LIN {X 0,Y 319.575,Z 275.493,A -85,B 0,C 180,E1 -15365.301,E2 -15365.301} C_VEL
LIN {X 0,Y 319.566,Z 275.493,A -85,B 0,C 180,E1 -15368.045,E2 -15368.045} C_VEL
LIN {X 0,Y 319.59,Z 275.527,A -85,B 0,C 180,E1 -15370.003,E2 -15370.003} C_VEL
LIN {X 0,Y 319.829,Z 276.598,A -85,B 0,C 180,E1 -15370.301,E2 -15370.301} C_VEL
LIN {X 0,Y 325.235,Z 292.198,A -85,B 0,C 180,E1 -15371.007,E2 -15371.007} C_VEL
LIN {X 0,Y 326.367,Z 298.329,A -85,B 0,C 180,E1 -15371.217,E2 -15371.217} C_VEL
LIN {X 0,Y 325.364,Z 352.937,A -85,B 0,C 180,E1 -15372.438,E2 -15372.438} C_VEL
LIN {X 0,Y 325.113,Z 362.734,A -85,B 0,C 180,E1 -15372.829,E2 -15372.829} C_VEL
LIN {X 0,Y 324.671,Z 373.811,A -85,B 0,C 180,E1 -15373.494,E2 -15373.494} C_VEL
LIN {X 0,Y 323.823,Z 384.617,A -85,B 0,C 180,E1 -15374.42,E2 -15374.42} C_VEL
LIN {X 0,Y 323.214,Z 391.764,A -85,B 0,C 180,E1 -15375.197,E2 -15375.197} C_VEL
LIN {X 0,Y 322.423,Z 399.87,A -85,B 0,C 180,E1 -15376.287,E2 -15376.287} C_VEL
LIN {X 0,Y 321.691,Z 406.556,A -85,B 0,C 180,E1 -15377.38,E2 -15377.38} C_VEL
LIN {X 0,Y 320.885,Z 412.887,A -85,B 0,C 180,E1 -15378.631,E2 -15378.631} C_VEL
LIN {X 0,Y 320.082,Z 419.308,A -85,B 0,C 180,E1 -15380.202,E2 -15380.202} C_VEL
LIN {X 0,Y 319.481,Z 424.66,A -85,B 0,C 180,E1 -15381.858,E2 -15381.858} C_VEL
LIN {X 0,Y 318.896,Z 429.161,A -85,B 0,C 180,E1 -15383.673,E2 -15383.673} C_VEL
LIN {X 0,Y 318.57,Z 431.47,A -85,B 0,C 180,E1 -15384.937,E2 -15384.937} C_VEL
LIN {X 0,Y 318.385,Z 433.223,A -85,B 0,C 180,E1 -15386.202,E2 -15386.202} C_VEL
LIN {X 0,Y 318.229,Z 434.488,A -85,B 0,C 180,E1 -15387.468,E2 -15387.468} C_VEL
LIN {X 0,Y 318.122,Z 435.287,A -85,B 0,C 180,E1 -15388.733,E2 -15388.733} C_VEL
LIN {X 0,Y 318.09,Z 435.591,A -85,B 0,C 180,E1 -15389.999,E2 -15389.999} C_VEL
LIN {X 0,Y 318.121,Z 435.315,A -85,B 0,C 180,E1 -15391.265,E2 -15391.265} C_VEL
LIN {X 0,Y 318.212,Z 434.573,A -85,B 0,C 180,E1 -15392.531,E2 -15392.531} C_VEL
LIN {X 0,Y 318.378,Z 433.365,A -85,B 0,C 180,E1 -15393.796,E2 -15393.796} C_VEL
LIN {X 0,Y 318.699,Z 430.531,A -85,B 0,C 180,E1 -15395.694,E2 -15395.694} C_VEL
LIN {X 0,Y 319.1,Z 427.945,A -85,B 0,C 180,E1 -15396.957,E2 -15396.957} C_VEL
LIN {X 0,Y 319.589,Z 424,A -85,B 0,C 180,E1 -15398.472,E2 -15398.472} C_VEL
LIN {X 0,Y 320.185,Z 418.558,A -85,B 0,C 180,E1 -15400.113,E2 -15400.113} C_VEL
LIN {X 0,Y 320.841,Z 413.383,A -85,B 0,C 180,E1 -15401.369,E2 -15401.369} C_VEL
LIN {X 0,Y 321.669,Z 407.142,A -85,B 0,C 180,E1 -15402.619,E2 -15402.619} C_VEL
LIN {X 0,Y 322.491,Z 399.559,A -85,B 0,C 180,E1 -15403.869,E2 -15403.869} C_VEL
LIN {X 0,Y 323.354,Z 390.109,A -85,B 0,C 180,E1 -15405.118,E2 -15405.118} C_VEL
LIN {X 0,Y 324.216,Z 380.839,A -85,B 0,C 180,E1 -15406.044,E2 -15406.044} C_VEL
LIN {X 0,Y 324.812,Z 371.887,A -85,B 0,C 180,E1 -15406.74,E2 -15406.74} C_VEL
LIN {X 0,Y 325.173,Z 362.547,A -85,B 0,C 180,E1 -15407.288,E2 -15407.288} C_VEL
LIN {X 0,Y 325.397,Z 353.548,A -85,B 0,C 180,E1 -15407.652,E2 -15407.652} C_VEL
LIN {X 0,Y 326.401,Z 302.241,A -85,B 0,C 180,E1 -15408.803,E2 -15408.803} C_VEL
LIN {X 0,Y 326.205,Z 297.195,A -85,B 0,C 180,E1 -15408.93,E2 -15408.93} C_VEL
LIN {X 0,Y 324.486,Z 289.724,A -85,B 0,C 180,E1 -15409.208,E2 -15409.208} C_VEL
LIN {X 0,Y 319.743,Z 276.336,A -85,B 0,C 180,E1 -15409.844,E2 -15409.844} C_VEL
LIN {X 0,Y 319.588,Z 275.493,A -85,B 0,C 180,E1 -15410.18,E2 -15410.18} C_VEL
LIN {X 0,Y 319.541,Z 275.494,A -85,B 0,C 180,E1 -15413.321,E2 -15413.321} C_VEL
LIN {X 0,Y 319.548,Z 275.494,A -85,B 0,C 180,E1 -15416.095,E2 -15416.095} C_VEL
LIN {X 0,Y 319.522,Z 275.496,A -85,B 0,C 180,E1 -15418.939,E2 -15418.939} C_VEL
LIN {X 0,Y 319.517,Z 275.496,A -85,B 0,C 180,E1 -15421.862,E2 -15421.862} C_VEL
LIN {X 0,Y 319.576,Z 275.487,A -85,B 0,C 180,E1 -15425.542,E2 -15425.542} C_VEL
LIN {X 0,Y 319.525,Z 275.495,A -85,B 0,C 180,E1 -15429.661,E2 -15429.661} C_VEL
LIN {X 0,Y 319.515,Z 275.495,A -85,B 0,C 180,E1 -15433.459,E2 -15433.459} C_VEL
LIN {X 0,Y 319.475,Z 275.497,A -85,B 0,C 180,E1 -15434.327,E2 -15434.327} C_VEL
LIN {X 0,Y 318.821,Z 275.583,A -85,B 0,C 180,E1 -15435.38,E2 -15435.38} C_VEL
LIN {X 0,Y 316.003,Z 275.942,A -85,B 0,C 180,E1 -15437.095,E2 -15437.095} C_VEL
LIN {X 0,Y 313.597,Z 276.243,A -85,B 0,C 180,E1 -15438.484,E2 -15438.484} C_VEL
LIN {X 0,Y 312.545,Z 276.369,A -85,B 0,C 180,E1 -15439.559,E2 -15439.559} C_VEL
LIN {X 0,Y 312.449,Z 276.378,A -85,B 0,C 180,E1 -15439.923,E2 -15439.923} C_VEL
LIN {X 0,Y 312.529,Z 276.366,A -85,B 0,C 180,E1 -15444.05,E2 -15444.05} C_VEL
LIN {X 0,Y 312.497,Z 276.371,A -85,B 0,C 180,E1 -15447.333,E2 -15447.333} C_VEL
LIN {X 0,Y 312.493,Z 276.373,A -85,B 0,C 180,E1 -15451.294,E2 -15451.294} C_VEL
LIN {X 0,Y 312.542,Z 276.364,A -85,B 0,C 180,E1 -15454.707,E2 -15454.707} C_VEL
LIN {X 0,Y 312.536,Z 276.367,A -85,B 0,C 180,E1 -15457.525,E2 -15457.525} C_VEL
LIN {X 0,Y 312.546,Z 276.363,A -85,B 0,C 180,E1 -15461.651,E2 -15461.651} C_VEL
LIN {X 0,Y 312.646,Z 276.346,A -85,B 0,C 180,E1 -15465.684,E2 -15465.684} C_VEL
LIN {X 0,Y 312.679,Z 276.346,A -85,B 0,C 180,E1 -15469.641,E2 -15469.641} C_VEL
LIN {X 0,Y 312.79,Z 276.333,A -85,B 0,C 180,E1 -15472.252,E2 -15472.252} C_VEL
LIN {X 0,Y 312.68,Z 276.345,A -85,B 0,C 180,E1 -15474.842,E2 -15474.842} C_VEL
LIN {X 0,Y 312.961,Z 276.313,A -85,B 0,C 180,E1 -15478.713,E2 -15478.713} C_VEL
LIN {X 0,Y 312.961,Z 276.311,A -85,B 0,C 180,E1 -15481.287,E2 -15481.287} C_VEL
LIN {X 0,Y 312.68,Z 276.345,A -85,B 0,C 180,E1 -15485.158,E2 -15485.158} C_VEL
LIN {X 0,Y 312.79,Z 276.333,A -85,B 0,C 180,E1 -15487.748,E2 -15487.748} C_VEL
LIN {X 0,Y 312.654,Z 276.349,A -85,B 0,C 180,E1 -15491.672,E2 -15491.672} C_VEL
LIN {X 0,Y 312.609,Z 276.355,A -85,B 0,C 180,E1 -15494.828,E2 -15494.828} C_VEL
LIN {X 0,Y 312.529,Z 276.365,A -85,B 0,C 180,E1 -15499.186,E2 -15499.186} C_VEL
LIN {X 0,Y 312.508,Z 276.368,A -85,B 0,C 180,E1 -15502.775,E2 -15502.775} C_VEL
LIN {X 0,Y 312.476,Z 276.372,A -85,B 0,C 180,E1 -15506.732,E2 -15506.732} C_VEL
LIN {X 0,Y 312.463,Z 276.379,A -85,B 0,C 180,E1 -15509.658,E2 -15509.658} C_VEL
LIN {X 0,Y 312.515,Z 276.372,A -85,B 0,C 180,E1 -15513.689,E2 -15513.689} C_VEL
LIN {X 0,Y 312.505,Z 276.374,A -85,B 0,C 180,E1 -15517.388,E2 -15517.388} C_VEL
LIN {X 0,Y 312.436,Z 276.378,A -85,B 0,C 180,E1 -15520.718,E2 -15520.718} C_VEL
LIN {X 0,Y 312.445,Z 276.376,A -85,B 0,C 180,E1 -15524.211,E2 -15524.211} C_VEL
LIN {X 0,Y 312.449,Z 276.376,A -85,B 0,C 180,E1 -15527.926,E2 -15527.926} C_VEL
LIN {X 0,Y 312.479,Z 276.372,A -85,B 0,C 180,E1 -15531.923,E2 -15531.923} C_VEL
LIN {X 0,Y 312.526,Z 276.366,A -85,B 0,C 180,E1 -15534.221,E2 -15534.221} C_VEL
LIN {X 0,Y 312.496,Z 276.371,A -85,B 0,C 180,E1 -15537.334,E2 -15537.334} C_VEL
LIN {X 0,Y 312.553,Z 276.446,A -85,B 0,C 180,E1 -15540.259,E2 -15540.259} C_VEL
LIN {X 0,Y 314.554,Z 286.634,A -85,B 0,C 180,E1 -15543.459,E2 -15543.459} C_VEL
LIN {X 0,Y 315.392,Z 291.548,A -85,B 0,C 180,E1 -15544.952,E2 -15544.952} C_VEL
LIN {X 0,Y 314.713,Z 298.783,A -85,B 0,C 180,E1 -15546.997,E2 -15546.997} C_VEL
LIN {X 0,Y 313.718,Z 308.843,A -85,B 0,C 180,E1 -15549.813,E2 -15549.813} C_VEL
LIN {X 0,Y 317.665,Z 337.125,A -85,B 0,C 180,E1 -15550.735,E2 -15550.735} C_VEL
LIN {X 0,Y 318.865,Z 349.16,A -85,B 0,C 180,E1 -15551.089,E2 -15551.089} C_VEL
LIN {X 0,Y 318.114,Z 387.635,A -85,B 0,C 180,E1 -15551.984,E2 -15551.984} C_VEL
LIN {X 0,Y 317.516,Z 398.812,A -85,B 0,C 180,E1 -15552.448,E2 -15552.448} C_VEL
LIN {X 0,Y 316.588,Z 410.517,A -85,B 0,C 180,E1 -15553.227,E2 -15553.227} C_VEL
LIN {X 0,Y 315.722,Z 419.221,A -85,B 0,C 180,E1 -15554.011,E2 -15554.011} C_VEL
LIN {X 0,Y 314.88,Z 427.545,A -85,B 0,C 180,E1 -15554.962,E2 -15554.962} C_VEL
LIN {X 0,Y 313.925,Z 435.427,A -85,B 0,C 180,E1 -15556.075,E2 -15556.075} C_VEL
LIN {X 0,Y 313.015,Z 442.804,A -85,B 0,C 180,E1 -15557.356,E2 -15557.356} C_VEL
LIN {X 0,Y 312.134,Z 450.298,A -85,B 0,C 180,E1 -15558.967,E2 -15558.967} C_VEL
LIN {X 0,Y 311.431,Z 457.151,A -85,B 0,C 180,E1 -15560.912,E2 -15560.912} C_VEL
LIN {X 0,Y 311.013,Z 462.366,A -85,B 0,C 180,E1 -15562.861,E2 -15562.861} C_VEL
LIN {X 0,Y 310.798,Z 466.2,A -85,B 0,C 180,E1 -15564.811,E2 -15564.811} C_VEL
LIN {X 0,Y 310.82,Z 467.97,A -85,B 0,C 180,E1 -15566.111,E2 -15566.111} C_VEL
LIN {X 0,Y 310.8,Z 469.234,A -85,B 0,C 180,E1 -15567.409,E2 -15567.409} C_VEL
LIN {X 0,Y 310.872,Z 470.023,A -85,B 0,C 180,E1 -15568.705,E2 -15568.705} C_VEL
LIN {X 0,Y 310.987,Z 470.326,A -85,B 0,C 180,E1 -15570.001,E2 -15570.001} C_VEL
LIN {X 0,Y 310.872,Z 470.018,A -85,B 0,C 180,E1 -15571.296,E2 -15571.296} C_VEL
LIN {X 0,Y 310.801,Z 469.217,A -85,B 0,C 180,E1 -15572.593,E2 -15572.593} C_VEL
LIN {X 0,Y 310.821,Z 467.941,A -85,B 0,C 180,E1 -15573.89,E2 -15573.89} C_VEL
LIN {X 0,Y 310.844,Z 464.997,A -85,B 0,C 180,E1 -15575.838,E2 -15575.838} C_VEL
LIN {X 0,Y 311.011,Z 462.314,A -85,B 0,C 180,E1 -15577.14,E2 -15577.14} C_VEL
LIN {X 0,Y 311.431,Z 457.083,A -85,B 0,C 180,E1 -15579.09,E2 -15579.09} C_VEL
LIN {X 0,Y 312.13,Z 450.197,A -85,B 0,C 180,E1 -15581.034,E2 -15581.034} C_VEL
LIN {X 0,Y 313.007,Z 442.688,A -85,B 0,C 180,E1 -15582.646,E2 -15582.646} C_VEL
LIN {X 0,Y 313.919,Z 435.29,A -85,B 0,C 180,E1 -15583.927,E2 -15583.927} C_VEL
LIN {X 0,Y 314.899,Z 427.377,A -85,B 0,C 180,E1 -15585.038,E2 -15585.038} C_VEL
LIN {X 0,Y 315.776,Z 419.013,A -85,B 0,C 180,E1 -15585.988,E2 -15585.988} C_VEL
LIN {X 0,Y 316.758,Z 408.327,A -85,B 0,C 180,E1 -15586.931,E2 -15586.931} C_VEL
LIN {X 0,Y 317.576,Z 396.677,A -85,B 0,C 180,E1 -15587.633,E2 -15587.633} C_VEL
LIN {X 0,Y 318.137,Z 386.897,A -85,B 0,C 180,E1 -15588.016,E2 -15588.016} C_VEL
LIN {X 0,Y 318.747,Z 347.007,A -85,B 0,C 180,E1 -15588.945,E2 -15588.945} C_VEL
LIN {X 0,Y 315.503,Z 321.052,A -85,B 0,C 180,E1 -15589.755,E2 -15589.755} C_VEL
LIN {X 0,Y 313.72,Z 308.721,A -85,B 0,C 180,E1 -15590.199,E2 -15590.199} C_VEL
LIN {X 0,Y 315.293,Z 293.881,A -85,B 0,C 180,E1 -15594.354,E2 -15594.354} C_VEL
LIN {X 0,Y 315.204,Z 290.232,A -85,B 0,C 180,E1 -15595.418,E2 -15595.418} C_VEL
LIN {X 0,Y 313.077,Z 279,A -85,B 0,C 180,E1 -15598.899,E2 -15598.899} C_VEL
LIN {X 0,Y 312.556,Z 276.361,A -85,B 0,C 180,E1 -15599.742,E2 -15599.742} C_VEL
LIN {X 0,Y 312.506,Z 276.367,A -85,B 0,C 180,E1 -15604.211,E2 -15604.211} C_VEL
LIN {X 0,Y 312.513,Z 276.37,A -85,B 0,C 180,E1 -15607.388,E2 -15607.388} C_VEL
LIN {X 0,Y 312.441,Z 276.38,A -85,B 0,C 180,E1 -15610.718,E2 -15610.718} C_VEL
LIN {X 0,Y 312.45,Z 276.376,A -85,B 0,C 180,E1 -15614.21,E2 -15614.21} C_VEL
LIN {X 0,Y 312.454,Z 276.375,A -85,B 0,C 180,E1 -15617.925,E2 -15617.925} C_VEL
LIN {X 0,Y 312.476,Z 276.373,A -85,B 0,C 180,E1 -15621.925,E2 -15621.925} C_VEL
LIN {X 0,Y 312.531,Z 276.368,A -85,B 0,C 180,E1 -15624.22,E2 -15624.22} C_VEL
LIN {X 0,Y 312.502,Z 276.368,A -85,B 0,C 180,E1 -15627.334,E2 -15627.334} C_VEL
LIN {X 0,Y 312.485,Z 276.37,A -85,B 0,C 180,E1 -15631.3,E2 -15631.3} C_VEL
LIN {X 0,Y 312.516,Z 276.368,A -85,B 0,C 180,E1 -15634.705,E2 -15634.705} C_VEL
LIN {X 0,Y 312.54,Z 276.364,A -85,B 0,C 180,E1 -15637.526,E2 -15637.526} C_VEL
LIN {X 0,Y 312.54,Z 276.366,A -85,B 0,C 180,E1 -15641.651,E2 -15641.651} C_VEL
LIN {X 0,Y 312.638,Z 276.354,A -85,B 0,C 180,E1 -15645.684,E2 -15645.684} C_VEL
LIN {X 0,Y 312.683,Z 276.348,A -85,B 0,C 180,E1 -15649.641,E2 -15649.641} C_VEL
LIN {X 0,Y 312.841,Z 276.324,A -85,B 0,C 180,E1 -15653.551,E2 -15653.551} C_VEL
LIN {X 0,Y 312.967,Z 276.31,A -85,B 0,C 180,E1 -15658.713,E2 -15658.713} C_VEL
LIN {X 0,Y 312.968,Z 276.313,A -85,B 0,C 180,E1 -15661.287,E2 -15661.287} C_VEL
LIN {X 0,Y 312.686,Z 276.343,A -85,B 0,C 180,E1 -15665.158,E2 -15665.158} C_VEL
LIN {X 0,Y 312.797,Z 276.332,A -85,B 0,C 180,E1 -15667.748,E2 -15667.748} C_VEL
LIN {X 0,Y 312.661,Z 276.348,A -85,B 0,C 180,E1 -15671.672,E2 -15671.672} C_VEL
LIN {X 0,Y 312.616,Z 276.352,A -85,B 0,C 180,E1 -15674.827,E2 -15674.827} C_VEL
LIN {X 0,Y 312.535,Z 276.367,A -85,B 0,C 180,E1 -15679.185,E2 -15679.185} C_VEL
LIN {X 0,Y 312.516,Z 276.37,A -85,B 0,C 180,E1 -15682.775,E2 -15682.775} C_VEL
LIN {X 0,Y 312.485,Z 276.374,A -85,B 0,C 180,E1 -15686.732,E2 -15686.732} C_VEL
LIN {X 0,Y 312.473,Z 276.371,A -85,B 0,C 180,E1 -15689.658,E2 -15689.658} C_VEL
LIN {X 0,Y 312.522,Z 276.364,A -85,B 0,C 180,E1 -15693.689,E2 -15693.689} C_VEL
LIN {X 0,Y 312.512,Z 276.366,A -85,B 0,C 180,E1 -15697.387,E2 -15697.387} C_VEL
LIN {X 0,Y 312.442,Z 276.376,A -85,B 0,C 180,E1 -15700.717,E2 -15700.717} C_VEL
LIN {X 0,Y 312.451,Z 276.379,A -85,B 0,C 180,E1 -15704.21,E2 -15704.21} C_VEL
LIN {X 0,Y 312.456,Z 276.378,A -85,B 0,C 180,E1 -15707.925,E2 -15707.925} C_VEL
LIN {X 0,Y 312.478,Z 276.365,A -85,B 0,C 180,E1 -15711.924,E2 -15711.924} C_VEL
LIN {X 0,Y 312.532,Z 276.365,A -85,B 0,C 180,E1 -15714.22,E2 -15714.22} C_VEL
LIN {X 0,Y 312.501,Z 276.371,A -85,B 0,C 180,E1 -15717.333,E2 -15717.333} C_VEL
LIN {X 0,Y 312.486,Z 276.373,A -85,B 0,C 180,E1 -15721.299,E2 -15721.299} C_VEL
LIN {X 0,Y 312.548,Z 276.365,A -85,B 0,C 180,E1 -15724.707,E2 -15724.707} C_VEL
LIN {X 0,Y 312.564,Z 276.368,A -85,B 0,C 180,E1 -15727.527,E2 -15727.527} C_VEL
LIN {X 0,Y 312.563,Z 276.573,A -85,B 0,C 180,E1 -15729.742,E2 -15729.742} C_VEL
LIN {X 0,Y 312.782,Z 277.421,A -85,B 0,C 180,E1 -15729.847,E2 -15729.847} C_VEL
LIN {X 0,Y 318.496,Z 293.396,A -85,B 0,C 180,E1 -15730.608,E2 -15730.608} C_VEL
LIN {X 0,Y 319.557,Z 298.349,A -85,B 0,C 180,E1 -15730.792,E2 -15730.792} C_VEL
LIN {X 0,Y 318.628,Z 353.345,A -85,B 0,C 180,E1 -15732.054,E2 -15732.054} C_VEL
LIN {X 0,Y 318.366,Z 363.135,A -85,B 0,C 180,E1 -15732.454,E2 -15732.454} C_VEL
LIN {X 0,Y 317.901,Z 374.209,A -85,B 0,C 180,E1 -15733.132,E2 -15733.132} C_VEL
LIN {X 0,Y 317.022,Z 385.012,A -85,B 0,C 180,E1 -15734.077,E2 -15734.077} C_VEL
LIN {X 0,Y 316.379,Z 392.158,A -85,B 0,C 180,E1 -15734.869,E2 -15734.869} C_VEL
LIN {X 0,Y 315.555,Z 400.265,A -85,B 0,C 180,E1 -15735.983,E2 -15735.983} C_VEL
LIN {X 0,Y 314.788,Z 406.95,A -85,B 0,C 180,E1 -15737.099,E2 -15737.099} C_VEL
LIN {X 0,Y 313.95,Z 413.28,A -85,B 0,C 180,E1 -15738.376,E2 -15738.376} C_VEL
LIN {X 0,Y 313.094,Z 419.702,A -85,B 0,C 180,E1 -15739.981,E2 -15739.981} C_VEL
LIN {X 0,Y 312.501,Z 424.818,A -85,B 0,C 180,E1 -15741.594,E2 -15741.594} C_VEL
LIN {X 0,Y 311.872,Z 429.552,A -85,B 0,C 180,E1 -15743.53,E2 -15743.53} C_VEL
LIN {X 0,Y 311.518,Z 431.862,A -85,B 0,C 180,E1 -15744.822,E2 -15744.822} C_VEL
LIN {X 0,Y 311.308,Z 433.615,A -85,B 0,C 180,E1 -15746.116,E2 -15746.116} C_VEL
LIN {X 0,Y 311.146,Z 434.88,A -85,B 0,C 180,E1 -15747.41,E2 -15747.41} C_VEL
LIN {X 0,Y 311.035,Z 435.679,A -85,B 0,C 180,E1 -15748.705,E2 -15748.705} C_VEL
LIN {X 0,Y 311.001,Z 435.983,A -85,B 0,C 180,E1 -15749.999,E2 -15749.999} C_VEL
LIN {X 0,Y 311.033,Z 435.707,A -85,B 0,C 180,E1 -15751.294,E2 -15751.294} C_VEL
LIN {X 0,Y 311.129,Z 434.964,A -85,B 0,C 180,E1 -15752.589,E2 -15752.589} C_VEL
LIN {X 0,Y 311.301,Z 433.756,A -85,B 0,C 180,E1 -15753.883,E2 -15753.883} C_VEL
LIN {X 0,Y 311.662,Z 430.921,A -85,B 0,C 180,E1 -15755.823,E2 -15755.823} C_VEL
LIN {X 0,Y 312.081,Z 428.334,A -85,B 0,C 180,E1 -15757.114,E2 -15757.114} C_VEL
LIN {X 0,Y 312.558,Z 424.529,A -85,B 0,C 180,E1 -15758.616,E2 -15758.616} C_VEL
LIN {X 0,Y 313.069,Z 420.11,A -85,B 0,C 180,E1 -15760.018,E2 -15760.018} C_VEL
LIN {X 0,Y 313.725,Z 415.181,A -85,B 0,C 180,E1 -15761.303,E2 -15761.303} C_VEL
LIN {X 0,Y 314.547,Z 409.224,A -85,B 0,C 180,E1 -15762.582,E2 -15762.582} C_VEL
LIN {X 0,Y 315.407,Z 401.975,A -85,B 0,C 180,E1 -15763.858,E2 -15763.858} C_VEL
LIN {X 0,Y 316.205,Z 394.225,A -85,B 0,C 180,E1 -15764.973,E2 -15764.973} C_VEL
LIN {X 0,Y 316.874,Z 387.535,A -85,B 0,C 180,E1 -15765.764,E2 -15765.764} C_VEL
LIN {X 0,Y 317.535,Z 379.358,A -85,B 0,C 180,E1 -15766.556,E2 -15766.556} C_VEL
LIN {X 0,Y 318.149,Z 371.061,A -85,B 0,C 180,E1 -15767.184,E2 -15767.184} C_VEL
LIN {X 0,Y 318.433,Z 362.098,A -85,B 0,C 180,E1 -15767.707,E2 -15767.707} C_VEL
LIN {X 0,Y 318.701,Z 352.449,A -85,B 0,C 180,E1 -15768.083,E2 -15768.083} C_VEL
LIN {X 0,Y 319.643,Z 298.831,A -85,B 0,C 180,E1 -15769.304,E2 -15769.304} C_VEL
LIN {X 0,Y 318.013,Z 291.836,A -85,B 0,C 180,E1 -15769.574,E2 -15769.574} C_VEL
LIN {X 0,Y 312.585,Z 276.757,A -85,B 0,C 180,E1 -15770.313,E2 -15770.313} C_VEL
LIN {X 0,Y 312.532,Z 276.374,A -85,B 0,C 180,E1 -15770.542,E2 -15770.542} C_VEL
LIN {X 0,Y 312.488,Z 276.372,A -85,B 0,C 180,E1 -15773.879,E2 -15773.879} C_VEL
LIN {X 0,Y 312.481,Z 276.376,A -85,B 0,C 180,E1 -15776.731,E2 -15776.731} C_VEL
LIN {X 0,Y 312.465,Z 276.374,A -85,B 0,C 180,E1 -15779.657,E2 -15779.657} C_VEL
LIN {X 0,Y 312.517,Z 276.367,A -85,B 0,C 180,E1 -15783.688,E2 -15783.688} C_VEL
LIN {X 0,Y 312.508,Z 276.367,A -85,B 0,C 180,E1 -15787.387,E2 -15787.387} C_VEL
LIN {X 0,Y 312.437,Z 276.375,A -85,B 0,C 180,E1 -15790.716,E2 -15790.716} C_VEL
LIN {X 0,Y 312.439,Z 276.378,A -85,B 0,C 180,E1 -15794.312,E2 -15794.312} C_VEL
LIN {X 0,Y 312.45,Z 276.375,A -85,B 0,C 180,E1 -15797.924,E2 -15797.924} C_VEL
LIN {X 0,Y 312.449,Z 276.378,A -85,B 0,C 180,E1 -15799.923,E2 -15799.923} C_VEL
LIN {X 0,Y 311.755,Z 276.462,A -85,B 0,C 180,E1 -15801,E2 -15801} C_VEL
LIN {X 0,Y 308.906,Z 276.815,A -85,B 0,C 180,E1 -15802.754,E2 -15802.754} C_VEL
LIN {X 0,Y 306.522,Z 277.114,A -85,B 0,C 180,E1 -15804.176,E2 -15804.176} C_VEL
LIN {X 0,Y 305.521,Z 277.239,A -85,B 0,C 180,E1 -15805.277,E2 -15805.277} C_VEL
LIN {X 0,Y 305.45,Z 277.247,A -85,B 0,C 180,E1 -15805.649,E2 -15805.649} C_VEL
LIN {X 0,Y 305.414,Z 277.256,A -85,B 0,C 180,E1 -15809.585,E2 -15809.585} C_VEL
LIN {X 0,Y 305.449,Z 277.245,A -85,B 0,C 180,E1 -15812.601,E2 -15812.601} C_VEL
LIN {X 0,Y 305.469,Z 277.247,A -85,B 0,C 180,E1 -15815.535,E2 -15815.535} C_VEL
LIN {X 0,Y 305.455,Z 277.245,A -85,B 0,C 180,E1 -15818.399,E2 -15818.399} C_VEL
LIN {X 0,Y 305.503,Z 277.244,A -85,B 0,C 180,E1 -15821.212,E2 -15821.212} C_VEL
LIN {X 0,Y 305.574,Z 277.228,A -85,B 0,C 180,E1 -15825.345,E2 -15825.345} C_VEL
LIN {X 0,Y 305.617,Z 277.227,A -85,B 0,C 180,E1 -15829.399,E2 -15829.399} C_VEL
LIN {X 0,Y 305.741,Z 277.21,A -85,B 0,C 180,E1 -15832.072,E2 -15832.072} C_VEL
LIN {X 0,Y 305.65,Z 277.22,A -85,B 0,C 180,E1 -15834.723,E2 -15834.723} C_VEL
LIN {X 0,Y 305.929,Z 277.188,A -85,B 0,C 180,E1 -15838.684,E2 -15838.684} C_VEL
LIN {X 0,Y 305.929,Z 277.187,A -85,B 0,C 180,E1 -15841.316,E2 -15841.316} C_VEL
LIN {X 0,Y 305.779,Z 277.209,A -85,B 0,C 180,E1 -15846.599,E2 -15846.599} C_VEL
LIN {X 0,Y 305.689,Z 277.216,A -85,B 0,C 180,E1 -15849.261,E2 -15849.261} C_VEL
LIN {X 0,Y 305.564,Z 277.233,A -85,B 0,C 180,E1 -15853.297,E2 -15853.297} C_VEL
LIN {X 0,Y 305.506,Z 277.243,A -85,B 0,C 180,E1 -15856.025,E2 -15856.025} C_VEL
LIN {X 0,Y 305.47,Z 277.247,A -85,B 0,C 180,E1 -15860.188,E2 -15860.188} C_VEL
LIN {X 0,Y 305.434,Z 277.249,A -85,B 0,C 180,E1 -15864.467,E2 -15864.467} C_VEL
LIN {X 0,Y 305.435,Z 277.252,A -85,B 0,C 180,E1 -15867.4,E2 -15867.4} C_VEL
LIN {X 0,Y 305.411,Z 277.253,A -85,B 0,C 180,E1 -15870.415,E2 -15870.415} C_VEL
LIN {X 0,Y 305.46,Z 277.248,A -85,B 0,C 180,E1 -15874.079,E2 -15874.079} C_VEL
LIN {X 0,Y 305.447,Z 277.249,A -85,B 0,C 180,E1 -15876.743,E2 -15876.743} C_VEL
LIN {X 0,Y 305.404,Z 277.254,A -85,B 0,C 180,E1 -15880.59,E2 -15880.59} C_VEL
LIN {X 0,Y 305.416,Z 277.254,A -85,B 0,C 180,E1 -15883.657,E2 -15883.657} C_VEL
LIN {X 0,Y 305.43,Z 277.253,A -85,B 0,C 180,E1 -15887.419,E2 -15887.419} C_VEL
LIN {X 0,Y 305.456,Z 277.248,A -85,B 0,C 180,E1 -15891.596,E2 -15891.596} C_VEL
LIN {X 0,Y 305.457,Z 277.25,A -85,B 0,C 180,E1 -15894.887,E2 -15894.887} C_VEL
LIN {X 0,Y 305.436,Z 277.251,A -85,B 0,C 180,E1 -15898.36,E2 -15898.36} C_VEL
LIN {X 0,Y 305.536,Z 277.384,A -85,B 0,C 180,E1 -15899.931,E2 -15899.931} C_VEL
LIN {X 0,Y 307.748,Z 288.821,A -85,B 0,C 180,E1 -15903.605,E2 -15903.605} C_VEL
LIN {X 0,Y 308.433,Z 293.564,A -85,B 0,C 180,E1 -15905.069,E2 -15905.069} C_VEL
LIN {X 0,Y 306.836,Z 308.508,A -85,B 0,C 180,E1 -15909.344,E2 -15909.344} C_VEL
LIN {X 0,Y 310.871,Z 337.091,A -85,B 0,C 180,E1 -15910.305,E2 -15910.305} C_VEL
LIN {X 0,Y 312.109,Z 350.383,A -85,B 0,C 180,E1 -15910.702,E2 -15910.702} C_VEL
LIN {X 0,Y 311.384,Z 387.259,A -85,B 0,C 180,E1 -15911.581,E2 -15911.581} C_VEL
LIN {X 0,Y 310.762,Z 398.43,A -85,B 0,C 180,E1 -15912.054,E2 -15912.054} C_VEL
LIN {X 0,Y 309.807,Z 410.131,A -85,B 0,C 180,E1 -15912.849,E2 -15912.849} C_VEL
LIN {X 0,Y 308.883,Z 418.832,A -85,B 0,C 180,E1 -15913.647,E2 -15913.647} C_VEL
LIN {X 0,Y 308.026,Z 427.157,A -85,B 0,C 180,E1 -15914.62,E2 -15914.62} C_VEL
LIN {X 0,Y 307.024,Z 435.037,A -85,B 0,C 180,E1 -15915.755,E2 -15915.755} C_VEL
LIN {X 0,Y 306.081,Z 442.414,A -85,B 0,C 180,E1 -15917.064,E2 -15917.064} C_VEL
LIN {X 0,Y 305.158,Z 449.907,A -85,B 0,C 180,E1 -15918.712,E2 -15918.712} C_VEL
LIN {X 0,Y 304.498,Z 455.792,A -85,B 0,C 180,E1 -15920.368,E2 -15920.368} C_VEL
LIN {X 0,Y 304.058,Z 460.437,A -85,B 0,C 180,E1 -15922.029,E2 -15922.029} C_VEL
LIN {X 0,Y 303.84,Z 463.46,A -85,B 0,C 180,E1 -15923.359,E2 -15923.359} C_VEL
LIN {X 0,Y 303.706,Z 465.808,A -85,B 0,C 180,E1 -15924.69,E2 -15924.69} C_VEL
LIN {X 0,Y 303.728,Z 467.578,A -85,B 0,C 180,E1 -15926.02,E2 -15926.02} C_VEL
LIN {X 0,Y 303.72,Z 468.843,A -85,B 0,C 180,E1 -15927.348,E2 -15927.348} C_VEL
LIN {X 0,Y 303.777,Z 469.632,A -85,B 0,C 180,E1 -15928.675,E2 -15928.675} C_VEL
LIN {X 0,Y 303.895,Z 469.934,A -85,B 0,C 180,E1 -15930.001,E2 -15930.001} C_VEL
LIN {X 0,Y 303.777,Z 469.626,A -85,B 0,C 180,E1 -15931.326,E2 -15931.326} C_VEL
LIN {X 0,Y 303.72,Z 468.825,A -85,B 0,C 180,E1 -15932.653,E2 -15932.653} C_VEL
LIN {X 0,Y 303.729,Z 467.548,A -85,B 0,C 180,E1 -15933.981,E2 -15933.981} C_VEL
LIN {X 0,Y 303.772,Z 464.865,A -85,B 0,C 180,E1 -15935.826,E2 -15935.826} C_VEL
LIN {X 0,Y 303.945,Z 461.92,A -85,B 0,C 180,E1 -15937.307,E2 -15937.307} C_VEL
LIN {X 0,Y 304.411,Z 456.689,A -85,B 0,C 180,E1 -15939.301,E2 -15939.301} C_VEL
LIN {X 0,Y 305.155,Z 449.803,A -85,B 0,C 180,E1 -15941.29,E2 -15941.29} C_VEL
LIN {X 0,Y 306.069,Z 442.292,A -85,B 0,C 180,E1 -15942.938,E2 -15942.938} C_VEL
LIN {X 0,Y 307.003,Z 434.894,A -85,B 0,C 180,E1 -15944.247,E2 -15944.247} C_VEL
LIN {X 0,Y 308.036,Z 426.981,A -85,B 0,C 180,E1 -15945.381,E2 -15945.381} C_VEL
LIN {X 0,Y 308.932,Z 418.615,A -85,B 0,C 180,E1 -15946.352,E2 -15946.352} C_VEL
LIN {X 0,Y 309.988,Z 407.929,A -85,B 0,C 180,E1 -15947.312,E2 -15947.312} C_VEL
LIN {X 0,Y 310.835,Z 396.277,A -85,B 0,C 180,E1 -15948.028,E2 -15948.028} C_VEL
LIN {X 0,Y 311.414,Z 386.491,A -85,B 0,C 180,E1 -15948.419,E2 -15948.419} C_VEL
LIN {X 0,Y 312.013,Z 347.585,A -85,B 0,C 180,E1 -15949.347,E2 -15949.347} C_VEL
LIN {X 0,Y 308.601,Z 320.295,A -85,B 0,C 180,E1 -15950.224,E2 -15950.224} C_VEL
LIN {X 0,Y 306.819,Z 308.34,A -85,B 0,C 180,E1 -15950.667,E2 -15950.667} C_VEL
LIN {X 0,Y 308.443,Z 293.47,A -85,B 0,C 180,E1 -15954.932,E2 -15954.932} C_VEL
LIN {X 0,Y 307.017,Z 284.868,A -85,B 0,C 180,E1 -15957.617,E2 -15957.617} C_VEL
LIN {X 0,Y 305.497,Z 277.238,A -85,B 0,C 180,E1 -15960.158,E2 -15960.158} C_VEL
LIN {X 0,Y 305.465,Z 277.244,A -85,B 0,C 180,E1 -15964.079,E2 -15964.079} C_VEL
LIN {X 0,Y 305.453,Z 277.249,A -85,B 0,C 180,E1 -15966.743,E2 -15966.743} C_VEL
LIN {X 0,Y 305.409,Z 277.255,A -85,B 0,C 180,E1 -15970.59,E2 -15970.59} C_VEL
LIN {X 0,Y 305.421,Z 277.251,A -85,B 0,C 180,E1 -15973.657,E2 -15973.657} C_VEL
LIN {X 0,Y 305.435,Z 277.25,A -85,B 0,C 180,E1 -15977.419,E2 -15977.419} C_VEL
LIN {X 0,Y 305.445,Z 277.248,A -85,B 0,C 180,E1 -15981.593,E2 -15981.593} C_VEL
LIN {X 0,Y 305.462,Z 277.248,A -85,B 0,C 180,E1 -15984.887,E2 -15984.887} C_VEL
LIN {X 0,Y 305.442,Z 277.252,A -85,B 0,C 180,E1 -15988.359,E2 -15988.359} C_VEL
LIN {X 0,Y 305.454,Z 277.246,A -85,B 0,C 180,E1 -15991.107,E2 -15991.107} C_VEL
LIN {X 0,Y 305.479,Z 277.247,A -85,B 0,C 180,E1 -15994.08,E2 -15994.08} C_VEL
LIN {X 0,Y 305.459,Z 277.248,A -85,B 0,C 180,E1 -15998.4,E2 -15998.4} C_VEL
LIN {X 0,Y 305.5,Z 277.241,A -85,B 0,C 180,E1 -16001.212,E2 -16001.212} C_VEL
LIN {X 0,Y 305.568,Z 277.233,A -85,B 0,C 180,E1 -16005.345,E2 -16005.345} C_VEL
LIN {X 0,Y 305.621,Z 277.226,A -85,B 0,C 180,E1 -16009.399,E2 -16009.399} C_VEL
LIN {X 0,Y 305.741,Z 277.205,A -85,B 0,C 180,E1 -16012.073,E2 -16012.073} C_VEL
LIN {X 0,Y 305.657,Z 277.218,A -85,B 0,C 180,E1 -16014.723,E2 -16014.723} C_VEL
LIN {X 0,Y 305.935,Z 277.186,A -85,B 0,C 180,E1 -16018.684,E2 -16018.684} C_VEL
LIN {X 0,Y 305.936,Z 277.187,A -85,B 0,C 180,E1 -16021.316,E2 -16021.316} C_VEL
LIN {X 0,Y 305.786,Z 277.203,A -85,B 0,C 180,E1 -16026.599,E2 -16026.599} C_VEL
LIN {X 0,Y 305.696,Z 277.22,A -85,B 0,C 180,E1 -16029.261,E2 -16029.261} C_VEL
LIN {X 0,Y 305.572,Z 277.229,A -85,B 0,C 180,E1 -16033.297,E2 -16033.297} C_VEL
LIN {X 0,Y 305.512,Z 277.233,A -85,B 0,C 180,E1 -16036.025,E2 -16036.025} C_VEL
LIN {X 0,Y 305.475,Z 277.244,A -85,B 0,C 180,E1 -16040.188,E2 -16040.188} C_VEL
LIN {X 0,Y 305.442,Z 277.25,A -85,B 0,C 180,E1 -16044.467,E2 -16044.467} C_VEL
LIN {X 0,Y 305.451,Z 277.246,A -85,B 0,C 180,E1 -16047.398,E2 -16047.398} C_VEL
LIN {X 0,Y 305.42,Z 277.254,A -85,B 0,C 180,E1 -16050.414,E2 -16050.414} C_VEL
LIN {X 0,Y 305.466,Z 277.244,A -85,B 0,C 180,E1 -16054.078,E2 -16054.078} C_VEL
LIN {X 0,Y 305.453,Z 277.248,A -85,B 0,C 180,E1 -16056.743,E2 -16056.743} C_VEL
LIN {X 0,Y 305.41,Z 277.253,A -85,B 0,C 180,E1 -16060.589,E2 -16060.589} C_VEL
LIN {X 0,Y 305.422,Z 277.249,A -85,B 0,C 180,E1 -16063.656,E2 -16063.656} C_VEL
LIN {X 0,Y 305.436,Z 277.25,A -85,B 0,C 180,E1 -16067.418,E2 -16067.418} C_VEL
LIN {X 0,Y 305.443,Z 277.239,A -85,B 0,C 180,E1 -16071.592,E2 -16071.592} C_VEL
LIN {X 0,Y 305.463,Z 277.244,A -85,B 0,C 180,E1 -16074.886,E2 -16074.886} C_VEL
LIN {X 0,Y 305.441,Z 277.249,A -85,B 0,C 180,E1 -16078.359,E2 -16078.359} C_VEL
LIN {X 0,Y 305.448,Z 277.248,A -85,B 0,C 180,E1 -16082.601,E2 -16082.601} C_VEL
LIN {X 0,Y 305.476,Z 277.251,A -85,B 0,C 180,E1 -16085.535,E2 -16085.535} C_VEL
LIN {X 0,Y 305.494,Z 277.25,A -85,B 0,C 180,E1 -16089.328,E2 -16089.328} C_VEL
LIN {X 0,Y 312.145,Z 295.838,A -85,B 0,C 180,E1 -16090.246,E2 -16090.246} C_VEL
LIN {X 0,Y 312.956,Z 300.347,A -85,B 0,C 180,E1 -16090.408,E2 -16090.408} C_VEL
LIN {X 0,Y 311.874,Z 352.463,A -85,B 0,C 180,E1 -16091.609,E2 -16091.609} C_VEL
LIN {X 0,Y 311.676,Z 361.879,A -85,B 0,C 180,E1 -16091.98,E2 -16091.98} C_VEL
LIN {X 0,Y 311.313,Z 371.012,A -85,B 0,C 180,E1 -16092.51,E2 -16092.51} C_VEL
LIN {X 0,Y 310.67,Z 380.336,A -85,B 0,C 180,E1 -16093.235,E2 -16093.235} C_VEL
LIN {X 0,Y 309.696,Z 389.897,A -85,B 0,C 180,E1 -16094.197,E2 -16094.197} C_VEL
LIN {X 0,Y 308.811,Z 399.644,A -85,B 0,C 180,E1 -16095.502,E2 -16095.502} C_VEL
LIN {X 0,Y 307.884,Z 407.344,A -85,B 0,C 180,E1 -16096.804,E2 -16096.804} C_VEL
LIN {X 0,Y 307.022,Z 413.673,A -85,B 0,C 180,E1 -16098.11,E2 -16098.11} C_VEL
LIN {X 0,Y 306.122,Z 420.095,A -85,B 0,C 180,E1 -16099.75,E2 -16099.75} C_VEL
LIN {X 0,Y 305.484,Z 425.212,A -85,B 0,C 180,E1 -16101.4,E2 -16101.4} C_VEL
LIN {X 0,Y 304.852,Z 429.943,A -85,B 0,C 180,E1 -16103.38,E2 -16103.38} C_VEL
LIN {X 0,Y 304.47,Z 432.254,A -85,B 0,C 180,E1 -16104.702,E2 -16104.702} C_VEL
LIN {X 0,Y 304.233,Z 434.008,A -85,B 0,C 180,E1 -16106.025,E2 -16106.025} C_VEL
LIN {X 0,Y 304.063,Z 435.272,A -85,B 0,C 180,E1 -16107.35,E2 -16107.35} C_VEL
LIN {X 0,Y 303.948,Z 436.07,A -85,B 0,C 180,E1 -16108.674,E2 -16108.674} C_VEL
LIN {X 0,Y 303.913,Z 436.374,A -85,B 0,C 180,E1 -16109.999,E2 -16109.999} C_VEL
LIN {X 0,Y 303.946,Z 436.098,A -85,B 0,C 180,E1 -16111.324,E2 -16111.324} C_VEL
LIN {X 0,Y 304.046,Z 435.355,A -85,B 0,C 180,E1 -16112.649,E2 -16112.649} C_VEL
LIN {X 0,Y 304.227,Z 434.147,A -85,B 0,C 180,E1 -16113.973,E2 -16113.973} C_VEL
LIN {X 0,Y 304.629,Z 431.31,A -85,B 0,C 180,E1 -16115.958,E2 -16115.958} C_VEL
LIN {X 0,Y 305.099,Z 428.154,A -85,B 0,C 180,E1 -16117.531,E2 -16117.531} C_VEL
LIN {X 0,Y 305.729,Z 423.642,A -85,B 0,C 180,E1 -16119.259,E2 -16119.259} C_VEL
LIN {X 0,Y 306.431,Z 418.172,A -85,B 0,C 180,E1 -16120.906,E2 -16120.906} C_VEL
LIN {X 0,Y 307.447,Z 411.285,A -85,B 0,C 180,E1 -16122.542,E2 -16122.542} C_VEL
LIN {X 0,Y 308.423,Z 403.378,A -85,B 0,C 180,E1 -16124.01,E2 -16124.01} C_VEL
LIN {X 0,Y 309.273,Z 395.833,A -85,B 0,C 180,E1 -16125.148,E2 -16125.148} C_VEL
LIN {X 0,Y 309.903,Z 389.417,A -85,B 0,C 180,E1 -16125.96,E2 -16125.96} C_VEL
LIN {X 0,Y 310.652,Z 381.607,A -85,B 0,C 180,E1 -16126.764,E2 -16126.764} C_VEL
LIN {X 0,Y 311.299,Z 372.651,A -85,B 0,C 180,E1 -16127.49,E2 -16127.49} C_VEL
LIN {X 0,Y 311.688,Z 363.306,A -85,B 0,C 180,E1 -16128.061,E2 -16128.061} C_VEL
LIN {X 0,Y 311.943,Z 353.774,A -85,B 0,C 180,E1 -16128.458,E2 -16128.458} C_VEL
LIN {X 0,Y 312.932,Z 299.702,A -85,B 0,C 180,E1 -16129.723,E2 -16129.723} C_VEL
LIN {X 0,Y 311.552,Z 293.883,A -85,B 0,C 180,E1 -16129.956,E2 -16129.956} C_VEL
LIN {X 0,Y 306.114,Z 279.394,A -85,B 0,C 180,E1 -16130.69,E2 -16130.69} C_VEL
LIN {X 0,Y 305.494,Z 277.251,A -85,B 0,C 180,E1 -16130.827,E2 -16130.827} C_VEL
LIN {X 0,Y 305.454,Z 277.251,A -85,B 0,C 180,E1 -16134.465,E2 -16134.465} C_VEL
LIN {X 0,Y 305.439,Z 277.25,A -85,B 0,C 180,E1 -16137.398,E2 -16137.398} C_VEL
LIN {X 0,Y 305.413,Z 277.256,A -85,B 0,C 180,E1 -16140.414,E2 -16140.414} C_VEL
LIN {X 0,Y 305.462,Z 277.249,A -85,B 0,C 180,E1 -16144.077,E2 -16144.077} C_VEL
LIN {X 0,Y 305.449,Z 277.247,A -85,B 0,C 180,E1 -16146.742,E2 -16146.742} C_VEL
LIN {X 0,Y 305.406,Z 277.251,A -85,B 0,C 180,E1 -16150.589,E2 -16150.589} C_VEL
LIN {X 0,Y 305.417,Z 277.252,A -85,B 0,C 180,E1 -16153.655,E2 -16153.655} C_VEL
LIN {X 0,Y 305.431,Z 277.248,A -85,B 0,C 180,E1 -16157.418,E2 -16157.418} C_VEL
LIN {X 0,Y 305.437,Z 277.251,A -85,B 0,C 180,E1 -16161.592,E2 -16161.592} C_VEL
LIN {X 0,Y 305.457,Z 277.245,A -85,B 0,C 180,E1 -16164.886,E2 -16164.886} C_VEL
LIN {X 0,Y 305.45,Z 277.247,A -85,B 0,C 180,E1 -16165.649,E2 -16165.649} C_VEL
LIN {X 0,Y 304.795,Z 277.332,A -85,B 0,C 180,E1 -16166.749,E2 -16166.749} C_VEL
LIN {X 0,Y 301.904,Z 277.691,A -85,B 0,C 180,E1 -16168.538,E2 -16168.538} C_VEL
LIN {X 0,Y 299.459,Z 277.994,A -85,B 0,C 180,E1 -16169.989,E2 -16169.989} C_VEL
LIN {X 0,Y 298.44,Z 278.122,A -85,B 0,C 180,E1 -16171.114,E2 -16171.114} C_VEL
LIN {X 0,Y 298.375,Z 278.126,A -85,B 0,C 180,E1 -16171.495,E2 -16171.495} C_VEL
LIN {X 0,Y 298.434,Z 278.122,A -85,B 0,C 180,E1 -16174.919,E2 -16174.919} C_VEL
LIN {X 0,Y 298.394,Z 278.126,A -85,B 0,C 180,E1 -16177.861,E2 -16177.861} C_VEL
LIN {X 0,Y 298.455,Z 278.12,A -85,B 0,C 180,E1 -16180.751,E2 -16180.751} C_VEL
LIN {X 0,Y 298.506,Z 278.107,A -85,B 0,C 180,E1 -16184.99,E2 -16184.99} C_VEL
LIN {X 0,Y 298.576,Z 278.106,A -85,B 0,C 180,E1 -16189.146,E2 -16189.146} C_VEL
LIN {X 0,Y 298.692,Z 278.088,A -85,B 0,C 180,E1 -16191.884,E2 -16191.884} C_VEL
LIN {X 0,Y 298.62,Z 278.096,A -85,B 0,C 180,E1 -16194.598,E2 -16194.598} C_VEL
LIN {X 0,Y 298.897,Z 278.063,A -85,B 0,C 180,E1 -16198.653,E2 -16198.653} C_VEL
LIN {X 0,Y 298.897,Z 278.063,A -85,B 0,C 180,E1 -16201.347,E2 -16201.347} C_VEL
LIN {X 0,Y 298.728,Z 278.086,A -85,B 0,C 180,E1 -16206.755,E2 -16206.755} C_VEL
LIN {X 0,Y 298.62,Z 278.097,A -85,B 0,C 180,E1 -16209.482,E2 -16209.482} C_VEL
LIN {X 0,Y 298.517,Z 278.112,A -85,B 0,C 180,E1 -16213.617,E2 -16213.617} C_VEL
LIN {X 0,Y 298.446,Z 278.122,A -85,B 0,C 180,E1 -16216.414,E2 -16216.414} C_VEL
LIN {X 0,Y 298.426,Z 278.124,A -85,B 0,C 180,E1 -16219.611,E2 -16219.611} C_VEL
LIN {X 0,Y 298.376,Z 278.131,A -85,B 0,C 180,E1 -16223.604,E2 -16223.604} C_VEL
LIN {X 0,Y 298.396,Z 278.126,A -85,B 0,C 180,E1 -16226.583,E2 -16226.583} C_VEL
LIN {X 0,Y 298.352,Z 278.136,A -85,B 0,C 180,E1 -16229.648,E2 -16229.648} C_VEL
LIN {X 0,Y 298.388,Z 278.128,A -85,B 0,C 180,E1 -16232.801,E2 -16232.801} C_VEL
LIN {X 0,Y 298.422,Z 278.124,A -85,B 0,C 180,E1 -16236.803,E2 -16236.803} C_VEL
LIN {X 0,Y 298.343,Z 278.136,A -85,B 0,C 180,E1 -16241.079,E2 -16241.079} C_VEL
LIN {X 0,Y 298.35,Z 278.136,A -85,B 0,C 180,E1 -16245.035,E2 -16245.035} C_VEL
LIN {X 0,Y 298.343,Z 278.137,A -85,B 0,C 180,E1 -16248.922,E2 -16248.922} C_VEL
LIN {X 0,Y 298.394,Z 278.127,A -85,B 0,C 180,E1 -16252.24,E2 -16252.24} C_VEL
LIN {X 0,Y 298.404,Z 278.126,A -85,B 0,C 180,E1 -16255.582,E2 -16255.582} C_VEL
LIN {X 0,Y 298.44,Z 278.181,A -85,B 0,C 180,E1 -16259.534,E2 -16259.534} C_VEL
LIN {X 0,Y 300.637,Z 289.286,A -85,B 0,C 180,E1 -16263.206,E2 -16263.206} C_VEL
LIN {X 0,Y 301.448,Z 294.361,A -85,B 0,C 180,E1 -16264.82,E2 -16264.82} C_VEL
LIN {X 0,Y 300.11,Z 306.38,A -85,B 0,C 180,E1 -16268.357,E2 -16268.357} C_VEL
LIN {X 0,Y 299.952,Z 308.023,A -85,B 0,C 180,E1 -16268.838,E2 -16268.838} C_VEL
LIN {X 0,Y 304.112,Z 337.152,A -85,B 0,C 180,E1 -16269.86,E2 -16269.86} C_VEL
LIN {X 0,Y 305.415,Z 349.86,A -85,B 0,C 180,E1 -16270.258,E2 -16270.258} C_VEL
LIN {X 0,Y 304.739,Z 385.968,A -85,B 0,C 180,E1 -16271.133,E2 -16271.133} C_VEL
LIN {X 0,Y 304.209,Z 395.232,A -85,B 0,C 180,E1 -16271.506,E2 -16271.506} C_VEL
LIN {X 0,Y 303.422,Z 405.687,A -85,B 0,C 180,E1 -16272.137,E2 -16272.137} C_VEL
LIN {X 0,Y 302.259,Z 416.94,A -85,B 0,C 180,E1 -16273.104,E2 -16273.104} C_VEL
LIN {X 0,Y 301.332,Z 425.534,A -85,B 0,C 180,E1 -16274.096,E2 -16274.096} C_VEL
LIN {X 0,Y 300.247,Z 433.62,A -85,B 0,C 180,E1 -16275.254,E2 -16275.254} C_VEL
LIN {X 0,Y 299.36,Z 440.309,A -85,B 0,C 180,E1 -16276.423,E2 -16276.423} C_VEL
LIN {X 0,Y 298.517,Z 446.664,A -85,B 0,C 180,E1 -16277.768,E2 -16277.768} C_VEL
LIN {X 0,Y 297.833,Z 451.95,A -85,B 0,C 180,E1 -16279.119,E2 -16279.119} C_VEL
LIN {X 0,Y 297.366,Z 456.367,A -85,B 0,C 180,E1 -16280.478,E2 -16280.478} C_VEL
LIN {X 0,Y 296.871,Z 461.581,A -85,B 0,C 180,E1 -16282.519,E2 -16282.519} C_VEL
LIN {X 0,Y 296.639,Z 465.417,A -85,B 0,C 180,E1 -16284.563,E2 -16284.563} C_VEL
LIN {X 0,Y 296.639,Z 467.186,A -85,B 0,C 180,E1 -16285.925,E2 -16285.925} C_VEL
LIN {X 0,Y 296.64,Z 468.452,A -85,B 0,C 180,E1 -16287.285,E2 -16287.285} C_VEL
LIN {X 0,Y 296.684,Z 469.24,A -85,B 0,C 180,E1 -16288.643,E2 -16288.643} C_VEL
LIN {X 0,Y 296.803,Z 469.543,A -85,B 0,C 180,E1 -16290.001,E2 -16290.001} C_VEL
LIN {X 0,Y 296.685,Z 469.234,A -85,B 0,C 180,E1 -16291.358,E2 -16291.358} C_VEL
LIN {X 0,Y 296.641,Z 468.434,A -85,B 0,C 180,E1 -16292.717,E2 -16292.717} C_VEL
LIN {X 0,Y 296.639,Z 467.155,A -85,B 0,C 180,E1 -16294.076,E2 -16294.076} C_VEL
LIN {X 0,Y 296.665,Z 464.849,A -85,B 0,C 180,E1 -16295.745,E2 -16295.745} C_VEL
LIN {X 0,Y 296.869,Z 461.525,A -85,B 0,C 180,E1 -16297.482,E2 -16297.482} C_VEL
LIN {X 0,Y 297.366,Z 456.293,A -85,B 0,C 180,E1 -16299.523,E2 -16299.523} C_VEL
LIN {X 0,Y 298.19,Z 449.408,A -85,B 0,C 180,E1 -16301.557,E2 -16301.557} C_VEL
LIN {X 0,Y 299.112,Z 441.895,A -85,B 0,C 180,E1 -16303.244,E2 -16303.244} C_VEL
LIN {X 0,Y 300.092,Z 434.497,A -85,B 0,C 180,E1 -16304.582,E2 -16304.582} C_VEL
LIN {X 0,Y 301.185,Z 426.584,A -85,B 0,C 180,E1 -16305.74,E2 -16305.74} C_VEL
LIN {X 0,Y 302.096,Z 418.217,A -85,B 0,C 180,E1 -16306.733,E2 -16306.733} C_VEL
LIN {X 0,Y 303.209,Z 407.586,A -85,B 0,C 180,E1 -16307.707,E2 -16307.707} C_VEL
LIN {X 0,Y 304.077,Z 396.36,A -85,B 0,C 180,E1 -16308.418,E2 -16308.418} C_VEL
LIN {X 0,Y 304.623,Z 387.32,A -85,B 0,C 180,E1 -16308.803,E2 -16308.803} C_VEL
LIN {X 0,Y 305.185,Z 360.313,A -85,B 0,C 180,E1 -16309.476,E2 -16309.476} C_VEL
LIN {X 0,Y 305.227,Z 347.515,A -85,B 0,C 180,E1 -16309.786,E2 -16309.786} C_VEL
LIN {X 0,Y 302.029,Z 321.952,A -85,B 0,C 180,E1 -16310.633,E2 -16310.633} C_VEL
LIN {X 0,Y 299.958,Z 307.909,A -85,B 0,C 180,E1 -16311.169,E2 -16311.169} C_VEL
LIN {X 0,Y 301.449,Z 294.264,A -85,B 0,C 180,E1 -16315.182,E2 -16315.182} C_VEL
LIN {X 0,Y 299.69,Z 284.422,A -85,B 0,C 180,E1 -16318.352,E2 -16318.352} C_VEL
LIN {X 0,Y 298.43,Z 278.119,A -85,B 0,C 180,E1 -16320.518,E2 -16320.518} C_VEL
LIN {X 0,Y 298.429,Z 278.121,A -85,B 0,C 180,E1 -16324.488,E2 -16324.488} C_VEL
LIN {X 0,Y 298.398,Z 278.126,A -85,B 0,C 180,E1 -16327.761,E2 -16327.761} C_VEL
LIN {X 0,Y 298.347,Z 278.135,A -85,B 0,C 180,E1 -16331.269,E2 -16331.269} C_VEL
LIN {X 0,Y 298.356,Z 278.135,A -85,B 0,C 180,E1 -16335.035,E2 -16335.035} C_VEL
LIN {X 0,Y 298.349,Z 278.136,A -85,B 0,C 180,E1 -16338.922,E2 -16338.922} C_VEL
LIN {X 0,Y 298.426,Z 278.123,A -85,B 0,C 180,E1 -16343.198,E2 -16343.198} C_VEL
LIN {X 0,Y 298.394,Z 278.126,A -85,B 0,C 180,E1 -16347.2,E2 -16347.2} C_VEL
LIN {X 0,Y 298.365,Z 278.132,A -85,B 0,C 180,E1 -16350.639,E2 -16350.639} C_VEL
LIN {X 0,Y 298.413,Z 278.124,A -85,B 0,C 180,E1 -16354.918,E2 -16354.918} C_VEL
LIN {X 0,Y 298.392,Z 278.129,A -85,B 0,C 180,E1 -16357.862,E2 -16357.862} C_VEL
LIN {X 0,Y 298.453,Z 278.119,A -85,B 0,C 180,E1 -16360.751,E2 -16360.751} C_VEL
LIN {X 0,Y 298.512,Z 278.111,A -85,B 0,C 180,E1 -16364.991,E2 -16364.991} C_VEL
LIN {X 0,Y 298.578,Z 278.102,A -85,B 0,C 180,E1 -16369.146,E2 -16369.146} C_VEL
LIN {X 0,Y 298.686,Z 278.083,A -85,B 0,C 180,E1 -16371.884,E2 -16371.884} C_VEL
LIN {X 0,Y 298.627,Z 278.093,A -85,B 0,C 180,E1 -16374.598,E2 -16374.598} C_VEL
LIN {X 0,Y 298.903,Z 278.062,A -85,B 0,C 180,E1 -16378.653,E2 -16378.653} C_VEL
LIN {X 0,Y 298.904,Z 278.062,A -85,B 0,C 180,E1 -16381.347,E2 -16381.347} C_VEL
LIN {X 0,Y 298.735,Z 278.081,A -85,B 0,C 180,E1 -16386.755,E2 -16386.755} C_VEL
LIN {X 0,Y 298.627,Z 278.099,A -85,B 0,C 180,E1 -16389.482,E2 -16389.482} C_VEL
LIN {X 0,Y 298.524,Z 278.104,A -85,B 0,C 180,E1 -16393.617,E2 -16393.617} C_VEL
LIN {X 0,Y 298.452,Z 278.113,A -85,B 0,C 180,E1 -16396.414,E2 -16396.414} C_VEL
LIN {X 0,Y 298.431,Z 278.121,A -85,B 0,C 180,E1 -16399.61,E2 -16399.61} C_VEL
LIN {X 0,Y 298.383,Z 278.126,A -85,B 0,C 180,E1 -16403.604,E2 -16403.604} C_VEL
LIN {X 0,Y 298.404,Z 278.129,A -85,B 0,C 180,E1 -16406.583,E2 -16406.583} C_VEL
LIN {X 0,Y 298.363,Z 278.129,A -85,B 0,C 180,E1 -16409.647,E2 -16409.647} C_VEL
LIN {X 0,Y 298.394,Z 278.125,A -85,B 0,C 180,E1 -16412.8,E2 -16412.8} C_VEL
LIN {X 0,Y 298.428,Z 278.122,A -85,B 0,C 180,E1 -16416.802,E2 -16416.802} C_VEL
LIN {X 0,Y 298.348,Z 278.13,A -85,B 0,C 180,E1 -16421.268,E2 -16421.268} C_VEL
LIN {X 0,Y 298.357,Z 278.131,A -85,B 0,C 180,E1 -16425.035,E2 -16425.035} C_VEL
LIN {X 0,Y 298.349,Z 278.128,A -85,B 0,C 180,E1 -16428.921,E2 -16428.921} C_VEL
LIN {X 0,Y 298.388,Z 278.117,A -85,B 0,C 180,E1 -16432.237,E2 -16432.237} C_VEL
LIN {X 0,Y 298.409,Z 278.126,A -85,B 0,C 180,E1 -16435.581,E2 -16435.581} C_VEL
LIN {X 0,Y 298.372,Z 278.129,A -85,B 0,C 180,E1 -16438.788,E2 -16438.788} C_VEL
LIN {X 0,Y 298.399,Z 278.129,A -85,B 0,C 180,E1 -16441.897,E2 -16441.897} C_VEL
LIN {X 0,Y 298.44,Z 278.124,A -85,B 0,C 180,E1 -16444.919,E2 -16444.919} C_VEL
LIN {X 0,Y 298.457,Z 278.125,A -85,B 0,C 180,E1 -16448.809,E2 -16448.809} C_VEL
LIN {X 0,Y 299.426,Z 280.925,A -85,B 0,C 180,E1 -16448.974,E2 -16448.974} C_VEL
LIN {X 0,Y 304.526,Z 294.377,A -85,B 0,C 180,E1 -16449.683,E2 -16449.683} C_VEL
LIN {X 0,Y 306.115,Z 300.014,A -85,B 0,C 180,E1 -16449.933,E2 -16449.933} C_VEL
LIN {X 0,Y 306.056,Z 313.052,A -85,B 0,C 180,E1 -16450.249,E2 -16450.249} C_VEL
LIN {X 0,Y 305.171,Z 352.871,A -85,B 0,C 180,E1 -16451.19,E2 -16451.19} C_VEL
LIN {X 0,Y 304.954,Z 362.282,A -85,B 0,C 180,E1 -16451.568,E2 -16451.568} C_VEL
LIN {X 0,Y 304.576,Z 371.411,A -85,B 0,C 180,E1 -16452.11,E2 -16452.11} C_VEL
LIN {X 0,Y 303.9,Z 380.734,A -85,B 0,C 180,E1 -16452.85,E2 -16452.85} C_VEL
LIN {X 0,Y 302.897,Z 390.293,A -85,B 0,C 180,E1 -16453.833,E2 -16453.833} C_VEL
LIN {X 0,Y 301.978,Z 400.037,A -85,B 0,C 180,E1 -16455.166,E2 -16455.166} C_VEL
LIN {X 0,Y 300.997,Z 407.738,A -85,B 0,C 180,E1 -16456.497,E2 -16456.497} C_VEL
LIN {X 0,Y 300.108,Z 414.066,A -85,B 0,C 180,E1 -16457.832,E2 -16457.832} C_VEL
LIN {X 0,Y 299.164,Z 420.487,A -85,B 0,C 180,E1 -16459.509,E2 -16459.509} C_VEL
LIN {X 0,Y 298.483,Z 425.604,A -85,B 0,C 180,E1 -16461.196,E2 -16461.196} C_VEL
LIN {X 0,Y 297.833,Z 430.335,A -85,B 0,C 180,E1 -16463.223,E2 -16463.223} C_VEL
LIN {X 0,Y 297.426,Z 432.645,A -85,B 0,C 180,E1 -16464.576,E2 -16464.576} C_VEL
LIN {X 0,Y 297.163,Z 434.4,A -85,B 0,C 180,E1 -16465.931,E2 -16465.931} C_VEL
LIN {X 0,Y 296.98,Z 435.664,A -85,B 0,C 180,E1 -16467.287,E2 -16467.287} C_VEL
LIN {X 0,Y 296.861,Z 436.462,A -85,B 0,C 180,E1 -16468.643,E2 -16468.643} C_VEL
LIN {X 0,Y 296.825,Z 436.766,A -85,B 0,C 180,E1 -16469.999,E2 -16469.999} C_VEL
LIN {X 0,Y 296.859,Z 436.489,A -85,B 0,C 180,E1 -16471.356,E2 -16471.356} C_VEL
LIN {X 0,Y 296.964,Z 435.746,A -85,B 0,C 180,E1 -16472.712,E2 -16472.712} C_VEL
LIN {X 0,Y 297.156,Z 434.537,A -85,B 0,C 180,E1 -16474.068,E2 -16474.068} C_VEL
LIN {X 0,Y 297.6,Z 431.699,A -85,B 0,C 180,E1 -16476.1,E2 -16476.1} C_VEL
LIN {X 0,Y 298.037,Z 428.854,A -85,B 0,C 180,E1 -16477.57,E2 -16477.57} C_VEL
LIN {X 0,Y 298.736,Z 424.032,A -85,B 0,C 180,E1 -16479.478,E2 -16479.478} C_VEL
LIN {X 0,Y 299.483,Z 418.561,A -85,B 0,C 180,E1 -16481.162,E2 -16481.162} C_VEL
LIN {X 0,Y 300.537,Z 411.674,A -85,B 0,C 180,E1 -16482.835,E2 -16482.835} C_VEL
LIN {X 0,Y 301.569,Z 403.764,A -85,B 0,C 180,E1 -16484.336,E2 -16484.336} C_VEL
LIN {X 0,Y 302.45,Z 396.22,A -85,B 0,C 180,E1 -16485.498,E2 -16485.498} C_VEL
LIN {X 0,Y 303.104,Z 389.802,A -85,B 0,C 180,E1 -16486.327,E2 -16486.327} C_VEL
LIN {X 0,Y 303.896,Z 381.991,A -85,B 0,C 180,E1 -16487.148,E2 -16487.148} C_VEL
LIN {X 0,Y 304.563,Z 373.033,A -85,B 0,C 180,E1 -16487.889,E2 -16487.889} C_VEL
LIN {X 0,Y 304.97,Z 363.685,A -85,B 0,C 180,E1 -16488.473,E2 -16488.473} C_VEL
LIN {X 0,Y 305.227,Z 354.996,A -85,B 0,C 180,E1 -16488.85,E2 -16488.85} C_VEL
LIN {X 0,Y 306.007,Z 319.979,A -85,B 0,C 180,E1 -16489.701,E2 -16489.701} C_VEL
LIN {X 0,Y 306.213,Z 300.356,A -85,B 0,C 180,E1 -16490.168,E2 -16490.168} C_VEL
LIN {X 0,Y 304.707,Z 294.872,A -85,B 0,C 180,E1 -16490.409,E2 -16490.409} C_VEL
LIN {X 0,Y 299.474,Z 280.995,A -85,B 0,C 180,E1 -16491.139,E2 -16491.139} C_VEL
LIN {X 0,Y 298.447,Z 278.128,A -85,B 0,C 180,E1 -16491.333,E2 -16491.333} C_VEL
LIN {X 0,Y 298.42,Z 278.127,A -85,B 0,C 180,E1 -16495.081,E2 -16495.081} C_VEL
LIN {X 0,Y 298.362,Z 278.131,A -85,B 0,C 180,E1 -16499.361,E2 -16499.361} C_VEL
LIN {X 0,Y 298.389,Z 278.128,A -85,B 0,C 180,E1 -16502.8,E2 -16502.8} C_VEL
LIN {X 0,Y 298.401,Z 278.126,A -85,B 0,C 180,E1 -16506.071,E2 -16506.071} C_VEL
LIN {X 0,Y 298.344,Z 278.133,A -85,B 0,C 180,E1 -16509.495,E2 -16509.495} C_VEL
LIN {X 0,Y 298.366,Z 278.128,A -85,B 0,C 180,E1 -16513.096,E2 -16513.096} C_VEL
LIN {X 0,Y 298.366,Z 278.126,A -85,B 0,C 180,E1 -16516.914,E2 -16516.914} C_VEL
LIN {X 0,Y 298.347,Z 278.131,A -85,B 0,C 180,E1 -16521.018,E2 -16521.018} C_VEL
LIN {X 0,Y 298.4,Z 278.127,A -85,B 0,C 180,E1 -16523.927,E2 -16523.927} C_VEL
LIN {X 0,Y 298.388,Z 278.127,A -85,B 0,C 180,E1 -16527.199,E2 -16527.199} C_VEL
LIN {X 0,Y 298.375,Z 278.126,A -85,B 0,C 180,E1 -16531.495,E2 -16531.495} C_VEL
LIN {X 0,Y 297.762,Z 278.206,A -85,B 0,C 180,E1 -16532.621,E2 -16532.621} C_VEL
LIN {X 0,Y 294.955,Z 278.562,A -85,B 0,C 180,E1 -16534.456,E2 -16534.456} C_VEL
LIN {X 0,Y 292.523,Z 278.865,A -85,B 0,C 180,E1 -16535.944,E2 -16535.944} C_VEL
LIN {X 0,Y 291.448,Z 278.994,A -85,B 0,C 180,E1 -16537.096,E2 -16537.096} C_VEL
LIN {X 0,Y 291.345,Z 279.005,A -85,B 0,C 180,E1 -16537.487,E2 -16537.487} C_VEL
LIN {X 0,Y 291.384,Z 278.999,A -85,B 0,C 180,E1 -16540.265,E2 -16540.265} C_VEL
LIN {X 0,Y 291.469,Z 278.984,A -85,B 0,C 180,E1 -16544.682,E2 -16544.682} C_VEL
LIN {X 0,Y 291.521,Z 278.984,A -85,B 0,C 180,E1 -16548.88,E2 -16548.88} C_VEL
LIN {X 0,Y 291.646,Z 278.966,A -85,B 0,C 180,E1 -16551.687,E2 -16551.687} C_VEL
LIN {X 0,Y 291.59,Z 278.972,A -85,B 0,C 180,E1 -16554.467,E2 -16554.467} C_VEL
LIN {X 0,Y 291.865,Z 278.937,A -85,B 0,C 180,E1 -16558.62,E2 -16558.62} C_VEL
LIN {X 0,Y 291.865,Z 278.939,A -85,B 0,C 180,E1 -16561.38,E2 -16561.38} C_VEL
LIN {X 0,Y 291.68,Z 278.963,A -85,B 0,C 180,E1 -16566.919,E2 -16566.919} C_VEL
LIN {X 0,Y 291.562,Z 278.977,A -85,B 0,C 180,E1 -16569.714,E2 -16569.714} C_VEL
LIN {X 0,Y 291.475,Z 278.991,A -85,B 0,C 180,E1 -16573.952,E2 -16573.952} C_VEL
LIN {X 0,Y 291.397,Z 278.998,A -85,B 0,C 180,E1 -16576.823,E2 -16576.823} C_VEL
LIN {X 0,Y 291.386,Z 279.002,A -85,B 0,C 180,E1 -16579.842,E2 -16579.842} C_VEL
LIN {X 0,Y 291.32,Z 279.008,A -85,B 0,C 180,E1 -16584.212,E2 -16584.212} C_VEL
LIN {X 0,Y 291.323,Z 279.009,A -85,B 0,C 180,E1 -16587.281,E2 -16587.281} C_VEL
LIN {X 0,Y 291.297,Z 279.011,A -85,B 0,C 180,E1 -16590.441,E2 -16590.441} C_VEL
LIN {X 0,Y 291.339,Z 279.01,A -85,B 0,C 180,E1 -16593.699,E2 -16593.699} C_VEL
LIN {X 0,Y 291.35,Z 279.008,A -85,B 0,C 180,E1 -16597.249,E2 -16597.249} C_VEL
LIN {X 0,Y 291.294,Z 279.012,A -85,B 0,C 180,E1 -16600.649,E2 -16600.649} C_VEL
LIN {X 0,Y 291.277,Z 279.014,A -85,B 0,C 180,E1 -16604.404,E2 -16604.404} C_VEL
LIN {X 0,Y 291.29,Z 279.012,A -85,B 0,C 180,E1 -16608.412,E2 -16608.412} C_VEL
LIN {X 0,Y 291.33,Z 279.01,A -85,B 0,C 180,E1 -16611.156,E2 -16611.156} C_VEL
LIN {X 0,Y 291.351,Z 279.007,A -85,B 0,C 180,E1 -16614.626,E2 -16614.626} C_VEL
LIN {X 0,Y 291.379,Z 279.123,A -85,B 0,C 180,E1 -16619.167,E2 -16619.167} C_VEL
LIN {X 0,Y 293.631,Z 290.247,A -85,B 0,C 180,E1 -16622.951,E2 -16622.951} C_VEL
LIN {X 0,Y 294.451,Z 295.158,A -85,B 0,C 180,E1 -16624.557,E2 -16624.557} C_VEL
LIN {X 0,Y 293.715,Z 302.382,A -85,B 0,C 180,E1 -16626.747,E2 -16626.747} C_VEL
LIN {X 0,Y 293.072,Z 307.598,A -85,B 0,C 180,E1 -16628.31,E2 -16628.31} C_VEL
LIN {X 0,Y 297.058,Z 334.539,A -85,B 0,C 180,E1 -16629.304,E2 -16629.304} C_VEL
LIN {X 0,Y 298.723,Z 350.377,A -85,B 0,C 180,E1 -16629.819,E2 -16629.819} C_VEL
LIN {X 0,Y 298.041,Z 385.582,A -85,B 0,C 180,E1 -16630.692,E2 -16630.692} C_VEL
LIN {X 0,Y 297.487,Z 395.023,A -85,B 0,C 180,E1 -16631.082,E2 -16631.082} C_VEL
LIN {X 0,Y 296.703,Z 404.681,A -85,B 0,C 180,E1 -16631.673,E2 -16631.673} C_VEL
LIN {X 0,Y 295.68,Z 414.96,A -85,B 0,C 180,E1 -16632.538,E2 -16632.538} C_VEL
LIN {X 0,Y 294.493,Z 425.145,A -85,B 0,C 180,E1 -16633.716,E2 -16633.716} C_VEL
LIN {X 0,Y 293.377,Z 433.231,A -85,B 0,C 180,E1 -16634.9,E2 -16634.9} C_VEL
LIN {X 0,Y 292.457,Z 439.919,A -85,B 0,C 180,E1 -16636.096,E2 -16636.096} C_VEL
LIN {X 0,Y 291.549,Z 446.273,A -85,B 0,C 180,E1 -16637.471,E2 -16637.471} C_VEL
LIN {X 0,Y 290.847,Z 451.559,A -85,B 0,C 180,E1 -16638.855,E2 -16638.855} C_VEL
LIN {X 0,Y 290.337,Z 455.975,A -85,B 0,C 180,E1 -16640.245,E2 -16640.245} C_VEL
LIN {X 0,Y 289.822,Z 461.19,A -85,B 0,C 180,E1 -16642.336,E2 -16642.336} C_VEL
LIN {X 0,Y 289.555,Z 465.025,A -85,B 0,C 180,E1 -16644.429,E2 -16644.429} C_VEL
LIN {X 0,Y 289.553,Z 466.794,A -85,B 0,C 180,E1 -16645.825,E2 -16645.825} C_VEL
LIN {X 0,Y 289.563,Z 468.061,A -85,B 0,C 180,E1 -16647.218,E2 -16647.218} C_VEL
LIN {X 0,Y 289.595,Z 468.849,A -85,B 0,C 180,E1 -16648.61,E2 -16648.61} C_VEL
LIN {X 0,Y 289.712,Z 469.151,A -85,B 0,C 180,E1 -16650.001,E2 -16650.001} C_VEL
LIN {X 0,Y 289.595,Z 468.842,A -85,B 0,C 180,E1 -16651.391,E2 -16651.391} C_VEL
LIN {X 0,Y 289.563,Z 468.042,A -85,B 0,C 180,E1 -16652.783,E2 -16652.783} C_VEL
LIN {X 0,Y 289.554,Z 466.762,A -85,B 0,C 180,E1 -16654.176,E2 -16654.176} C_VEL
LIN {X 0,Y 289.626,Z 463.814,A -85,B 0,C 180,E1 -16656.269,E2 -16656.269} C_VEL
LIN {X 0,Y 289.82,Z 461.131,A -85,B 0,C 180,E1 -16657.665,E2 -16657.665} C_VEL
LIN {X 0,Y 290.338,Z 455.898,A -85,B 0,C 180,E1 -16659.756,E2 -16659.756} C_VEL
LIN {X 0,Y 291.223,Z 449.013,A -85,B 0,C 180,E1 -16661.838,E2 -16661.838} C_VEL
LIN {X 0,Y 292.181,Z 441.499,A -85,B 0,C 180,E1 -16663.564,E2 -16663.564} C_VEL
LIN {X 0,Y 293.217,Z 434.101,A -85,B 0,C 180,E1 -16664.932,E2 -16664.932} C_VEL
LIN {X 0,Y 294.332,Z 426.187,A -85,B 0,C 180,E1 -16666.116,E2 -16666.116} C_VEL
LIN {X 0,Y 295.295,Z 417.82,A -85,B 0,C 180,E1 -16667.13,E2 -16667.13} C_VEL
LIN {X 0,Y 296.427,Z 407.379,A -85,B 0,C 180,E1 -16668.11,E2 -16668.11} C_VEL
LIN {X 0,Y 297.354,Z 396.191,A -85,B 0,C 180,E1 -16668.837,E2 -16668.837} C_VEL
LIN {X 0,Y 297.93,Z 386.776,A -85,B 0,C 180,E1 -16669.247,E2 -16669.247} C_VEL
LIN {X 0,Y 298.59,Z 355.979,A -85,B 0,C 180,E1 -16670.023,E2 -16670.023} C_VEL
LIN {X 0,Y 298.539,Z 348.297,A -85,B 0,C 180,E1 -16670.218,E2 -16670.218} C_VEL
LIN {X 0,Y 295.482,Z 323.431,A -85,B 0,C 180,E1 -16671.064,E2 -16671.064} C_VEL
LIN {X 0,Y 293.151,Z 307.508,A -85,B 0,C 180,E1 -16671.686,E2 -16671.686} C_VEL
LIN {X 0,Y 294.414,Z 296.843,A -85,B 0,C 180,E1 -16674.892,E2 -16674.892} C_VEL
LIN {X 0,Y 294.276,Z 293.835,A -85,B 0,C 180,E1 -16675.84,E2 -16675.84} C_VEL
LIN {X 0,Y 292.301,Z 283.399,A -85,B 0,C 180,E1 -16679.321,E2 -16679.321} C_VEL
LIN {X 0,Y 291.371,Z 279,A -85,B 0,C 180,E1 -16680.885,E2 -16680.885} C_VEL
LIN {X 0,Y 291.355,Z 279.006,A -85,B 0,C 180,E1 -16685.375,E2 -16685.375} C_VEL
LIN {X 0,Y 291.334,Z 279.01,A -85,B 0,C 180,E1 -16688.845,E2 -16688.845} C_VEL
LIN {X 0,Y 291.287,Z 279.014,A -85,B 0,C 180,E1 -16692.499,E2 -16692.499} C_VEL
LIN {X 0,Y 291.289,Z 279.014,A -85,B 0,C 180,E1 -16696.371,E2 -16696.371} C_VEL
LIN {X 0,Y 291.313,Z 279.013,A -85,B 0,C 180,E1 -16700.535,E2 -16700.535} C_VEL
LIN {X 0,Y 291.387,Z 279.002,A -85,B 0,C 180,E1 -16702.917,E2 -16702.917} C_VEL
LIN {X 0,Y 291.345,Z 279.008,A -85,B 0,C 180,E1 -16706.302,E2 -16706.302} C_VEL
LIN {X 0,Y 291.336,Z 279.01,A -85,B 0,C 180,E1 -16710.279,E2 -16710.279} C_VEL
LIN {X 0,Y 291.343,Z 279.009,A -85,B 0,C 180,E1 -16714.265,E2 -16714.265} C_VEL
LIN {X 0,Y 291.35,Z 279.004,A -85,B 0,C 180,E1 -16717.297,E2 -16717.297} C_VEL
LIN {X 0,Y 291.386,Z 279.002,A -85,B 0,C 180,E1 -16720.265,E2 -16720.265} C_VEL
LIN {X 0,Y 291.453,Z 278.99,A -85,B 0,C 180,E1 -16724.699,E2 -16724.699} C_VEL
LIN {X 0,Y 291.523,Z 278.98,A -85,B 0,C 180,E1 -16728.88,E2 -16728.88} C_VEL
LIN {X 0,Y 291.632,Z 278.961,A -85,B 0,C 180,E1 -16731.686,E2 -16731.686} C_VEL
LIN {X 0,Y 291.597,Z 278.969,A -85,B 0,C 180,E1 -16734.468,E2 -16734.468} C_VEL
LIN {X 0,Y 291.87,Z 278.938,A -85,B 0,C 180,E1 -16738.62,E2 -16738.62} C_VEL
LIN {X 0,Y 291.872,Z 278.936,A -85,B 0,C 180,E1 -16741.38,E2 -16741.38} C_VEL
LIN {X 0,Y 291.687,Z 278.96,A -85,B 0,C 180,E1 -16746.919,E2 -16746.919} C_VEL
LIN {X 0,Y 291.57,Z 278.977,A -85,B 0,C 180,E1 -16749.714,E2 -16749.714} C_VEL
LIN {X 0,Y 291.483,Z 278.979,A -85,B 0,C 180,E1 -16753.952,E2 -16753.952} C_VEL
LIN {X 0,Y 291.403,Z 278.993,A -85,B 0,C 180,E1 -16756.823,E2 -16756.823} C_VEL
LIN {X 0,Y 291.393,Z 278.998,A -85,B 0,C 180,E1 -16759.842,E2 -16759.842} C_VEL
LIN {X 0,Y 291.328,Z 279.006,A -85,B 0,C 180,E1 -16764.212,E2 -16764.212} C_VEL
LIN {X 0,Y 291.334,Z 279.004,A -85,B 0,C 180,E1 -16767.281,E2 -16767.281} C_VEL
LIN {X 0,Y 291.306,Z 279.013,A -85,B 0,C 180,E1 -16770.441,E2 -16770.441} C_VEL
LIN {X 0,Y 291.345,Z 279,A -85,B 0,C 180,E1 -16773.698,E2 -16773.698} C_VEL
LIN {X 0,Y 291.354,Z 279.002,A -85,B 0,C 180,E1 -16777.247,E2 -16777.247} C_VEL
LIN {X 0,Y 291.296,Z 279.009,A -85,B 0,C 180,E1 -16781.588,E2 -16781.588} C_VEL
LIN {X 0,Y 291.284,Z 279.014,A -85,B 0,C 180,E1 -16785.596,E2 -16785.596} C_VEL
LIN {X 0,Y 291.301,Z 279.007,A -85,B 0,C 180,E1 -16789.351,E2 -16789.351} C_VEL
LIN {X 0,Y 291.387,Z 278.989,A -85,B 0,C 180,E1 -16792.916,E2 -16792.916} C_VEL
LIN {X 0,Y 291.345,Z 279.005,A -85,B 0,C 180,E1 -16796.301,E2 -16796.301} C_VEL
LIN {X 0,Y 291.336,Z 279.007,A -85,B 0,C 180,E1 -16800.278,E2 -16800.278} C_VEL
LIN {X 0,Y 291.36,Z 279.006,A -85,B 0,C 180,E1 -16804.266,E2 -16804.266} C_VEL
LIN {X 0,Y 291.399,Z 279.005,A -85,B 0,C 180,E1 -16808.282,E2 -16808.282} C_VEL
LIN {X 0,Y 292.865,Z 283.041,A -85,B 0,C 180,E1 -16808.524,E2 -16808.524} C_VEL
LIN {X 0,Y 297.407,Z 294.444,A -85,B 0,C 180,E1 -16809.164,E2 -16809.164} C_VEL
LIN {X 0,Y 299.605,Z 301.665,A -85,B 0,C 180,E1 -16809.509,E2 -16809.509} C_VEL
LIN {X 0,Y 298.49,Z 354.571,A -85,B 0,C 180,E1 -16810.798,E2 -16810.798} C_VEL
LIN {X 0,Y 298.189,Z 364.342,A -85,B 0,C 180,E1 -16811.224,E2 -16811.224} C_VEL
LIN {X 0,Y 297.668,Z 375.403,A -85,B 0,C 180,E1 -16811.947,E2 -16811.947} C_VEL
LIN {X 0,Y 296.666,Z 386.2,A -85,B 0,C 180,E1 -16812.952,E2 -16812.952} C_VEL
LIN {X 0,Y 295.914,Z 393.344,A -85,B 0,C 180,E1 -16813.795,E2 -16813.795} C_VEL
LIN {X 0,Y 294.981,Z 401.448,A -85,B 0,C 180,E1 -16814.983,E2 -16814.983} C_VEL
LIN {X 0,Y 294.123,Z 408.131,A -85,B 0,C 180,E1 -16816.175,E2 -16816.175} C_VEL
LIN {X 0,Y 293.18,Z 414.46,A -85,B 0,C 180,E1 -16817.54,E2 -16817.54} C_VEL
LIN {X 0,Y 292.199,Z 420.88,A -85,B 0,C 180,E1 -16819.256,E2 -16819.256} C_VEL
LIN {X 0,Y 291.483,Z 425.995,A -85,B 0,C 180,E1 -16820.983,E2 -16820.983} C_VEL
LIN {X 0,Y 290.812,Z 430.726,A -85,B 0,C 180,E1 -16823.059,E2 -16823.059} C_VEL
LIN {X 0,Y 290.386,Z 433.037,A -85,B 0,C 180,E1 -16824.444,E2 -16824.444} C_VEL
LIN {X 0,Y 290.097,Z 434.791,A -85,B 0,C 180,E1 -16825.831,E2 -16825.831} C_VEL
LIN {X 0,Y 289.898,Z 436.055,A -85,B 0,C 180,E1 -16827.22,E2 -16827.22} C_VEL
LIN {X 0,Y 289.774,Z 436.853,A -85,B 0,C 180,E1 -16828.61,E2 -16828.61} C_VEL
LIN {X 0,Y 289.736,Z 437.157,A -85,B 0,C 180,E1 -16829.999,E2 -16829.999} C_VEL
LIN {X 0,Y 289.772,Z 436.88,A -85,B 0,C 180,E1 -16831.389,E2 -16831.389} C_VEL
LIN {X 0,Y 289.882,Z 436.137,A -85,B 0,C 180,E1 -16832.779,E2 -16832.779} C_VEL
LIN {X 0,Y 290.09,Z 434.928,A -85,B 0,C 180,E1 -16834.167,E2 -16834.167} C_VEL
LIN {X 0,Y 290.574,Z 432.089,A -85,B 0,C 180,E1 -16836.248,E2 -16836.248} C_VEL
LIN {X 0,Y 290.973,Z 429.558,A -85,B 0,C 180,E1 -16837.609,E2 -16837.609} C_VEL
LIN {X 0,Y 291.736,Z 424.422,A -85,B 0,C 180,E1 -16839.708,E2 -16839.708} C_VEL
LIN {X 0,Y 292.521,Z 418.951,A -85,B 0,C 180,E1 -16841.432,E2 -16841.432} C_VEL
LIN {X 0,Y 293.633,Z 412.062,A -85,B 0,C 180,E1 -16843.142,E2 -16843.142} C_VEL
LIN {X 0,Y 294.727,Z 404.151,A -85,B 0,C 180,E1 -16844.676,E2 -16844.676} C_VEL
LIN {X 0,Y 295.639,Z 396.606,A -85,B 0,C 180,E1 -16845.865,E2 -16845.865} C_VEL
LIN {X 0,Y 296.319,Z 390.188,A -85,B 0,C 180,E1 -16846.712,E2 -16846.712} C_VEL
LIN {X 0,Y 297.153,Z 382.374,A -85,B 0,C 180,E1 -16847.55,E2 -16847.55} C_VEL
LIN {X 0,Y 297.842,Z 373.415,A -85,B 0,C 180,E1 -16848.307,E2 -16848.307} C_VEL
LIN {X 0,Y 298.273,Z 364.064,A -85,B 0,C 180,E1 -16848.903,E2 -16848.903} C_VEL
LIN {X 0,Y 298.528,Z 355.483,A -85,B 0,C 180,E1 -16849.286,E2 -16849.286} C_VEL
LIN {X 0,Y 299.338,Z 323.008,A -85,B 0,C 180,E1 -16850.092,E2 -16850.092} C_VEL
LIN {X 0,Y 299.596,Z 301.392,A -85,B 0,C 180,E1 -16850.616,E2 -16850.616} C_VEL
LIN {X 0,Y 295.18,Z 288.422,A -85,B 0,C 180,E1 -16851.277,E2 -16851.277} C_VEL
LIN {X 0,Y 291.48,Z 279.677,A -85,B 0,C 180,E1 -16851.794,E2 -16851.794} C_VEL
LIN {X 0,Y 291.362,Z 279.011,A -85,B 0,C 180,E1 -16851.862,E2 -16851.862} C_VEL
LIN {X 0,Y 291.345,Z 279.008,A -85,B 0,C 180,E1 -16855.734,E2 -16855.734} C_VEL
LIN {X 0,Y 291.332,Z 279.007,A -85,B 0,C 180,E1 -16859.72,E2 -16859.72} C_VEL
LIN {X 0,Y 291.341,Z 279.005,A -85,B 0,C 180,E1 -16863.698,E2 -16863.698} C_VEL
LIN {X 0,Y 291.35,Z 279.002,A -85,B 0,C 180,E1 -16867.247,E2 -16867.247} C_VEL
LIN {X 0,Y 291.291,Z 279.008,A -85,B 0,C 180,E1 -16871.588,E2 -16871.588} C_VEL
LIN {X 0,Y 291.279,Z 279.014,A -85,B 0,C 180,E1 -16875.596,E2 -16875.596} C_VEL
LIN {X 0,Y 291.29,Z 279.007,A -85,B 0,C 180,E1 -16879.35,E2 -16879.35} C_VEL
LIN {X 0,Y 291.382,Z 278.998,A -85,B 0,C 180,E1 -16882.916,E2 -16882.916} C_VEL
LIN {X 0,Y 291.34,Z 279.004,A -85,B 0,C 180,E1 -16886.301,E2 -16886.301} C_VEL
LIN {X 0,Y 291.334,Z 279.005,A -85,B 0,C 180,E1 -16890.277,E2 -16890.277} C_VEL
LIN {X 0,Y 291.353,Z 279.003,A -85,B 0,C 180,E1 -16894.266,E2 -16894.266} C_VEL
LIN {X 0,Y 291.345,Z 279.005,A -85,B 0,C 180,E1 -16897.487,E2 -16897.487} C_VEL
LIN {X 0,Y 290.635,Z 279.093,A -85,B 0,C 180,E1 -16898.641,E2 -16898.641} C_VEL
LIN {X 0,Y 287.777,Z 279.449,A -85,B 0,C 180,E1 -16900.521,E2 -16900.521} C_VEL
LIN {X 0,Y 285.401,Z 279.743,A -85,B 0,C 180,E1 -16902.048,E2 -16902.048} C_VEL
LIN {X 0,Y 284.415,Z 279.864,A -85,B 0,C 180,E1 -16903.23,E2 -16903.23} C_VEL
LIN {X 0,Y 284.35,Z 279.868,A -85,B 0,C 180,E1 -16903.63,E2 -16903.63} C_VEL
LIN {X 0,Y 284.452,Z 279.861,A -85,B 0,C 180,E1 -16907.152,E2 -16907.152} C_VEL
LIN {X 0,Y 284.603,Z 279.844,A -85,B 0,C 180,E1 -16911.479,E2 -16911.479} C_VEL
LIN {X 0,Y 284.561,Z 279.847,A -85,B 0,C 180,E1 -16914.33,E2 -16914.33} C_VEL
LIN {X 0,Y 284.832,Z 279.812,A -85,B 0,C 180,E1 -16918.586,E2 -16918.586} C_VEL
LIN {X 0,Y 284.832,Z 279.815,A -85,B 0,C 180,E1 -16921.414,E2 -16921.414} C_VEL
LIN {X 0,Y 284.636,Z 279.84,A -85,B 0,C 180,E1 -16927.091,E2 -16927.091} C_VEL
LIN {X 0,Y 284.508,Z 279.857,A -85,B 0,C 180,E1 -16929.957,E2 -16929.957} C_VEL
LIN {X 0,Y 284.412,Z 279.87,A -85,B 0,C 180,E1 -16934.306,E2 -16934.306} C_VEL
LIN {X 0,Y 284.312,Z 279.88,A -85,B 0,C 180,E1 -16938.745,E2 -16938.745} C_VEL
LIN {X 0,Y 284.292,Z 279.886,A -85,B 0,C 180,E1 -16941.766,E2 -16941.766} C_VEL
LIN {X 0,Y 284.278,Z 279.883,A -85,B 0,C 180,E1 -16944.852,E2 -16944.852} C_VEL
LIN {X 0,Y 284.254,Z 279.891,A -85,B 0,C 180,E1 -16948.019,E2 -16948.019} C_VEL
LIN {X 0,Y 284.273,Z 279.888,A -85,B 0,C 180,E1 -16951.277,E2 -16951.277} C_VEL
LIN {X 0,Y 284.332,Z 279.883,A -85,B 0,C 180,E1 -16955.347,E2 -16955.347} C_VEL
LIN {X 0,Y 284.262,Z 279.888,A -85,B 0,C 180,E1 -16958.177,E2 -16958.177} C_VEL
LIN {X 0,Y 284.232,Z 279.892,A -85,B 0,C 180,E1 -16962.117,E2 -16962.117} C_VEL
LIN {X 0,Y 284.233,Z 279.892,A -85,B 0,C 180,E1 -16966.186,E2 -16966.186} C_VEL
LIN {X 0,Y 284.279,Z 279.885,A -85,B 0,C 180,E1 -16970.03,E2 -16970.03} C_VEL
LIN {X 0,Y 284.317,Z 279.881,A -85,B 0,C 180,E1 -16973.613,E2 -16973.613} C_VEL
LIN {X 0,Y 284.316,Z 279.88,A -85,B 0,C 180,E1 -16977.897,E2 -16977.897} C_VEL
LIN {X 0,Y 284.341,Z 279.911,A -85,B 0,C 180,E1 -16978.732,E2 -16978.732} C_VEL
LIN {X 0,Y 286.576,Z 291.038,A -85,B 0,C 180,E1 -16982.625,E2 -16982.625} C_VEL
LIN {X 0,Y 287.481,Z 296.403,A -85,B 0,C 180,E1 -16984.427,E2 -16984.427} C_VEL
LIN {X 0,Y 286.753,Z 303.177,A -85,B 0,C 180,E1 -16986.531,E2 -16986.531} C_VEL
LIN {X 0,Y 286.235,Z 307.192,A -85,B 0,C 180,E1 -16987.764,E2 -16987.764} C_VEL
LIN {X 0,Y 290.097,Z 332.937,A -85,B 0,C 180,E1 -16988.752,E2 -16988.752} C_VEL
LIN {X 0,Y 292.048,Z 350.879,A -85,B 0,C 180,E1 -16989.359,E2 -16989.359} C_VEL
LIN {X 0,Y 291.298,Z 386.132,A -85,B 0,C 180,E1 -16990.26,E2 -16990.26} C_VEL
LIN {X 0,Y 290.612,Z 397.3,A -85,B 0,C 180,E1 -16990.763,E2 -16990.763} C_VEL
LIN {X 0,Y 289.525,Z 408.972,A -85,B 0,C 180,E1 -16991.606,E2 -16991.606} C_VEL
LIN {X 0,Y 288.514,Z 417.669,A -85,B 0,C 180,E1 -16992.456,E2 -16992.456} C_VEL
LIN {X 0,Y 287.487,Z 425.988,A -85,B 0,C 180,E1 -16993.49,E2 -16993.49} C_VEL
LIN {X 0,Y 286.365,Z 433.866,A -85,B 0,C 180,E1 -16994.704,E2 -16994.704} C_VEL
LIN {X 0,Y 285.284,Z 441.241,A -85,B 0,C 180,E1 -16996.103,E2 -16996.103} C_VEL
LIN {X 0,Y 284.239,Z 448.734,A -85,B 0,C 180,E1 -16997.869,E2 -16997.869} C_VEL
LIN {X 0,Y 283.285,Z 455.581,A -85,B 0,C 180,E1 -17000,E2 -17000} C_VEL
LIN {X 0,Y 282.756,Z 460.797,A -85,B 0,C 180,E1 -17002.144,E2 -17002.144} C_VEL
LIN {X 0,Y 282.484,Z 464.757,A -85,B 0,C 180,E1 -17004.366,E2 -17004.366} C_VEL
LIN {X 0,Y 282.452,Z 466.402,A -85,B 0,C 180,E1 -17005.72,E2 -17005.72} C_VEL
LIN {X 0,Y 282.487,Z 467.67,A -85,B 0,C 180,E1 -17007.149,E2 -17007.149} C_VEL
LIN {X 0,Y 282.509,Z 468.457,A -85,B 0,C 180,E1 -17008.575,E2 -17008.575} C_VEL
LIN {X 0,Y 282.62,Z 468.76,A -85,B 0,C 180,E1 -17010.001,E2 -17010.001} C_VEL
LIN {X 0,Y 282.509,Z 468.451,A -85,B 0,C 180,E1 -17011.426,E2 -17011.426} C_VEL
LIN {X 0,Y 282.487,Z 467.651,A -85,B 0,C 180,E1 -17012.853,E2 -17012.853} C_VEL
LIN {X 0,Y 282.453,Z 466.369,A -85,B 0,C 180,E1 -17014.282,E2 -17014.282} C_VEL
LIN {X 0,Y 282.567,Z 463.42,A -85,B 0,C 180,E1 -17016.427,E2 -17016.427} C_VEL
LIN {X 0,Y 282.754,Z 460.736,A -85,B 0,C 180,E1 -17017.858,E2 -17017.858} C_VEL
LIN {X 0,Y 283.285,Z 455.501,A -85,B 0,C 180,E1 -17020.002,E2 -17020.002} C_VEL
LIN {X 0,Y 284.237,Z 448.617,A -85,B 0,C 180,E1 -17022.133,E2 -17022.133} C_VEL
LIN {X 0,Y 285.272,Z 441.104,A -85,B 0,C 180,E1 -17023.899,E2 -17023.899} C_VEL
LIN {X 0,Y 286.361,Z 433.706,A -85,B 0,C 180,E1 -17025.298,E2 -17025.298} C_VEL
LIN {X 0,Y 287.496,Z 425.79,A -85,B 0,C 180,E1 -17026.51,E2 -17026.51} C_VEL
LIN {X 0,Y 288.509,Z 417.423,A -85,B 0,C 180,E1 -17027.545,E2 -17027.545} C_VEL
LIN {X 0,Y 289.664,Z 407.168,A -85,B 0,C 180,E1 -17028.531,E2 -17028.531} C_VEL
LIN {X 0,Y 290.651,Z 395.507,A -85,B 0,C 180,E1 -17029.304,E2 -17029.304} C_VEL
LIN {X 0,Y 291.249,Z 386.512,A -85,B 0,C 180,E1 -17029.701,E2 -17029.701} C_VEL
LIN {X 0,Y 291.876,Z 358.146,A -85,B 0,C 180,E1 -17030.437,E2 -17030.437} C_VEL
LIN {X 0,Y 291.92,Z 349.449,A -85,B 0,C 180,E1 -17030.658,E2 -17030.658} C_VEL
LIN {X 0,Y 288.949,Z 324.96,A -85,B 0,C 180,E1 -17031.513,E2 -17031.513} C_VEL
LIN {X 0,Y 286.27,Z 307.162,A -85,B 0,C 180,E1 -17032.213,E2 -17032.213} C_VEL
LIN {X 0,Y 287.468,Z 297.368,A -85,B 0,C 180,E1 -17035.234,E2 -17035.234} C_VEL
LIN {X 0,Y 286.783,Z 292.163,A -85,B 0,C 180,E1 -17036.961,E2 -17036.961} C_VEL
LIN {X 0,Y 284.68,Z 281.483,A -85,B 0,C 180,E1 -17040.669,E2 -17040.669} C_VEL
LIN {X 0,Y 284.344,Z 279.874,A -85,B 0,C 180,E1 -17041.269,E2 -17041.269} C_VEL
LIN {X 0,Y 284.337,Z 279.88,A -85,B 0,C 180,E1 -17045.347,E2 -17045.347} C_VEL
LIN {X 0,Y 284.298,Z 279.883,A -85,B 0,C 180,E1 -17048.172,E2 -17048.172} C_VEL
LIN {X 0,Y 284.237,Z 279.891,A -85,B 0,C 180,E1 -17052.117,E2 -17052.117} C_VEL
LIN {X 0,Y 284.238,Z 279.891,A -85,B 0,C 180,E1 -17056.186,E2 -17056.186} C_VEL
LIN {X 0,Y 284.257,Z 279.889,A -85,B 0,C 180,E1 -17060.037,E2 -17060.037} C_VEL
LIN {X 0,Y 284.319,Z 279.88,A -85,B 0,C 180,E1 -17063.612,E2 -17063.612} C_VEL
LIN {X 0,Y 284.307,Z 279.881,A -85,B 0,C 180,E1 -17067.191,E2 -17067.191} C_VEL
LIN {X 0,Y 284.31,Z 279.885,A -85,B 0,C 180,E1 -17070.371,E2 -17070.371} C_VEL
LIN {X 0,Y 284.296,Z 279.883,A -85,B 0,C 180,E1 -17073.579,E2 -17073.579} C_VEL
LIN {X 0,Y 284.309,Z 279.882,A -85,B 0,C 180,E1 -17076.702,E2 -17076.702} C_VEL
LIN {X 0,Y 284.335,Z 279.88,A -85,B 0,C 180,E1 -17079.928,E2 -17079.928} C_VEL
LIN {X 0,Y 284.422,Z 279.866,A -85,B 0,C 180,E1 -17084.513,E2 -17084.513} C_VEL
LIN {X 0,Y 284.453,Z 279.86,A -85,B 0,C 180,E1 -17088.6,E2 -17088.6} C_VEL
LIN {X 0,Y 284.583,Z 279.839,A -85,B 0,C 180,E1 -17091.479,E2 -17091.479} C_VEL
LIN {X 0,Y 284.567,Z 279.844,A -85,B 0,C 180,E1 -17094.331,E2 -17094.331} C_VEL
LIN {X 0,Y 284.837,Z 279.814,A -85,B 0,C 180,E1 -17098.586,E2 -17098.586} C_VEL
LIN {X 0,Y 284.839,Z 279.811,A -85,B 0,C 180,E1 -17101.414,E2 -17101.414} C_VEL
LIN {X 0,Y 284.643,Z 279.838,A -85,B 0,C 180,E1 -17107.092,E2 -17107.092} C_VEL
LIN {X 0,Y 284.516,Z 279.855,A -85,B 0,C 180,E1 -17109.957,E2 -17109.957} C_VEL
LIN {X 0,Y 284.42,Z 279.859,A -85,B 0,C 180,E1 -17114.306,E2 -17114.306} C_VEL
LIN {X 0,Y 284.318,Z 279.88,A -85,B 0,C 180,E1 -17118.744,E2 -17118.744} C_VEL
LIN {X 0,Y 284.298,Z 279.881,A -85,B 0,C 180,E1 -17121.766,E2 -17121.766} C_VEL
LIN {X 0,Y 284.285,Z 279.887,A -85,B 0,C 180,E1 -17124.852,E2 -17124.852} C_VEL
LIN {X 0,Y 284.267,Z 279.885,A -85,B 0,C 180,E1 -17128.018,E2 -17128.018} C_VEL
LIN {X 0,Y 284.281,Z 279.884,A -85,B 0,C 180,E1 -17131.276,E2 -17131.276} C_VEL
LIN {X 0,Y 284.338,Z 279.87,A -85,B 0,C 180,E1 -17135.346,E2 -17135.346} C_VEL
LIN {X 0,Y 284.265,Z 279.889,A -85,B 0,C 180,E1 -17138.177,E2 -17138.177} C_VEL
LIN {X 0,Y 284.238,Z 279.888,A -85,B 0,C 180,E1 -17142.117,E2 -17142.117} C_VEL
LIN {X 0,Y 284.24,Z 279.894,A -85,B 0,C 180,E1 -17146.185,E2 -17146.185} C_VEL
LIN {X 0,Y 284.285,Z 279.874,A -85,B 0,C 180,E1 -17150.029,E2 -17150.029} C_VEL
LIN {X 0,Y 284.32,Z 279.871,A -85,B 0,C 180,E1 -17153.612,E2 -17153.612} C_VEL
LIN {X 0,Y 284.307,Z 279.882,A -85,B 0,C 180,E1 -17157.19,E2 -17157.19} C_VEL
LIN {X 0,Y 284.31,Z 279.882,A -85,B 0,C 180,E1 -17160.37,E2 -17160.37} C_VEL
LIN {X 0,Y 284.304,Z 279.887,A -85,B 0,C 180,E1 -17163.579,E2 -17163.579} C_VEL
LIN {X 0,Y 284.345,Z 279.886,A -85,B 0,C 180,E1 -17167.747,E2 -17167.747} C_VEL
LIN {X 0,Y 285.278,Z 282.603,A -85,B 0,C 180,E1 -17167.898,E2 -17167.898} C_VEL
LIN {X 0,Y 290.396,Z 294.967,A -85,B 0,C 180,E1 -17168.639,E2 -17168.639} C_VEL
LIN {X 0,Y 293.003,Z 303.183,A -85,B 0,C 180,E1 -17169.054,E2 -17169.054} C_VEL
LIN {X 0,Y 291.802,Z 353.688,A -85,B 0,C 180,E1 -17170.294,E2 -17170.294} C_VEL
LIN {X 0,Y 291.559,Z 363.086,A -85,B 0,C 180,E1 -17170.689,E2 -17170.689} C_VEL
LIN {X 0,Y 291.151,Z 372.208,A -85,B 0,C 180,E1 -17171.255,E2 -17171.255} C_VEL
LIN {X 0,Y 290.434,Z 381.526,A -85,B 0,C 180,E1 -17172.029,E2 -17172.029} C_VEL
LIN {X 0,Y 289.337,Z 391.084,A -85,B 0,C 180,E1 -17173.053,E2 -17173.053} C_VEL
LIN {X 0,Y 288.315,Z 400.826,A -85,B 0,C 180,E1 -17174.446,E2 -17174.446} C_VEL
LIN {X 0,Y 287.258,Z 408.525,A -85,B 0,C 180,E1 -17175.838,E2 -17175.838} C_VEL
LIN {X 0,Y 286.277,Z 414.853,A -85,B 0,C 180,E1 -17177.235,E2 -17177.235} C_VEL
LIN {X 0,Y 285.236,Z 421.274,A -85,B 0,C 180,E1 -17178.991,E2 -17178.991} C_VEL
LIN {X 0,Y 284.478,Z 426.389,A -85,B 0,C 180,E1 -17180.759,E2 -17180.759} C_VEL
LIN {X 0,Y 283.794,Z 431.118,A -85,B 0,C 180,E1 -17182.887,E2 -17182.887} C_VEL
LIN {X 0,Y 283.35,Z 433.428,A -85,B 0,C 180,E1 -17184.305,E2 -17184.305} C_VEL
LIN {X 0,Y 283.034,Z 435.183,A -85,B 0,C 180,E1 -17185.727,E2 -17185.727} C_VEL
LIN {X 0,Y 282.819,Z 436.447,A -85,B 0,C 180,E1 -17187.151,E2 -17187.151} C_VEL
LIN {X 0,Y 282.688,Z 437.245,A -85,B 0,C 180,E1 -17188.575,E2 -17188.575} C_VEL
LIN {X 0,Y 282.648,Z 437.548,A -85,B 0,C 180,E1 -17189.999,E2 -17189.999} C_VEL
LIN {X 0,Y 282.685,Z 437.272,A -85,B 0,C 180,E1 -17191.424,E2 -17191.424} C_VEL
LIN {X 0,Y 282.803,Z 436.528,A -85,B 0,C 180,E1 -17192.848,E2 -17192.848} C_VEL
LIN {X 0,Y 283.027,Z 435.318,A -85,B 0,C 180,E1 -17194.271,E2 -17194.271} C_VEL
LIN {X 0,Y 283.552,Z 432.478,A -85,B 0,C 180,E1 -17196.403,E2 -17196.403} C_VEL
LIN {X 0,Y 284.153,Z 428.717,A -85,B 0,C 180,E1 -17198.378,E2 -17198.378} C_VEL
LIN {X 0,Y 285.043,Z 422.828,A -85,B 0,C 180,E1 -17200.656,E2 -17200.656} C_VEL
LIN {X 0,Y 286.019,Z 416.734,A -85,B 0,C 180,E1 -17202.415,E2 -17202.415} C_VEL
LIN {X 0,Y 287.021,Z 410.774,A -85,B 0,C 180,E1 -17203.811,E2 -17203.811} C_VEL
LIN {X 0,Y 288.008,Z 403.524,A -85,B 0,C 180,E1 -17205.207,E2 -17205.207} C_VEL
LIN {X 0,Y 288.953,Z 395.771,A -85,B 0,C 180,E1 -17206.423,E2 -17206.423} C_VEL
LIN {X 0,Y 289.734,Z 389.077,A -85,B 0,C 180,E1 -17207.285,E2 -17207.285} C_VEL
LIN {X 0,Y 290.537,Z 380.894,A -85,B 0,C 180,E1 -17208.145,E2 -17208.145} C_VEL
LIN {X 0,Y 291.251,Z 372.59,A -85,B 0,C 180,E1 -17208.828,E2 -17208.828} C_VEL
LIN {X 0,Y 291.604,Z 363.615,A -85,B 0,C 180,E1 -17209.398,E2 -17209.398} C_VEL
LIN {X 0,Y 291.884,Z 354.813,A -85,B 0,C 180,E1 -17209.78,E2 -17209.78} C_VEL
LIN {X 0,Y 293.067,Z 302.861,A -85,B 0,C 180,E1 -17211.069,E2 -17211.069} C_VEL
LIN {X 0,Y 288.072,Z 289.029,A -85,B 0,C 180,E1 -17211.823,E2 -17211.823} C_VEL
LIN {X 0,Y 284.472,Z 280.733,A -85,B 0,C 180,E1 -17212.342,E2 -17212.342} C_VEL
LIN {X 0,Y 284.303,Z 279.892,A -85,B 0,C 180,E1 -17212.422,E2 -17212.422} C_VEL
LIN {X 0,Y 284.295,Z 279.887,A -85,B 0,C 180,E1 -17216.421,E2 -17216.421} C_VEL
LIN {X 0,Y 284.271,Z 279.888,A -85,B 0,C 180,E1 -17220.083,E2 -17220.083} C_VEL
LIN {X 0,Y 284.302,Z 279.882,A -85,B 0,C 180,E1 -17222.945,E2 -17222.945} C_VEL
LIN {X 0,Y 284.316,Z 279.88,A -85,B 0,C 180,E1 -17226.387,E2 -17226.387} C_VEL
LIN {X 0,Y 284.252,Z 279.89,A -85,B 0,C 180,E1 -17230.003,E2 -17230.003} C_VEL
LIN {X 0,Y 284.231,Z 279.893,A -85,B 0,C 180,E1 -17234.187,E2 -17234.187} C_VEL
LIN {X 0,Y 284.235,Z 279.886,A -85,B 0,C 180,E1 -17238.118,E2 -17238.118} C_VEL
LIN {X 0,Y 284.277,Z 279.884,A -85,B 0,C 180,E1 -17242.288,E2 -17242.288} C_VEL
LIN {X 0,Y 284.303,Z 279.882,A -85,B 0,C 180,E1 -17245.35,E2 -17245.35} C_VEL
LIN {X 0,Y 284.274,Z 279.883,A -85,B 0,C 180,E1 -17248.723,E2 -17248.723} C_VEL
LIN {X 0,Y 284.323,Z 279.876,A -85,B 0,C 180,E1 -17252.854,E2 -17252.854} C_VEL
LIN {X 0,Y 284.322,Z 279.879,A -85,B 0,C 180,E1 -17256.703,E2 -17256.703} C_VEL
LIN {X 0,Y 284.318,Z 279.881,A -85,B 0,C 180,E1 -17261.256,E2 -17261.256} C_VEL
LIN {X 0,Y 284.35,Z 279.868,A -85,B 0,C 180,E1 -17263.63,E2 -17263.63} C_VEL
LIN {X 0,Y 283.725,Z 279.946,A -85,B 0,C 180,E1 -17264.812,E2 -17264.812} C_VEL
LIN {X 0,Y 280.901,Z 280.301,A -85,B 0,C 180,E1 -17266.738,E2 -17266.738} C_VEL
LIN {X 0,Y 278.507,Z 280.602,A -85,B 0,C 180,E1 -17268.303,E2 -17268.303} C_VEL
LIN {X 0,Y 277.516,Z 280.728,A -85,B 0,C 180,E1 -17269.516,E2 -17269.516} C_VEL
LIN {X 0,Y 277.456,Z 280.734,A -85,B 0,C 180,E1 -17269.926,E2 -17269.926} C_VEL
LIN {X 0,Y 277.595,Z 280.718,A -85,B 0,C 180,E1 -17272.727,E2 -17272.727} C_VEL
LIN {X 0,Y 277.799,Z 280.687,A -85,B 0,C 180,E1 -17278.55,E2 -17278.55} C_VEL
LIN {X 0,Y 277.799,Z 280.691,A -85,B 0,C 180,E1 -17281.45,E2 -17281.45} C_VEL
LIN {X 0,Y 277.594,Z 280.717,A -85,B 0,C 180,E1 -17287.272,E2 -17287.272} C_VEL
LIN {X 0,Y 277.448,Z 280.736,A -85,B 0,C 180,E1 -17290.213,E2 -17290.213} C_VEL
LIN {X 0,Y 277.365,Z 280.745,A -85,B 0,C 180,E1 -17294.678,E2 -17294.678} C_VEL
LIN {X 0,Y 277.271,Z 280.757,A -85,B 0,C 180,E1 -17299.239,E2 -17299.239} C_VEL
LIN {X 0,Y 277.25,Z 280.762,A -85,B 0,C 180,E1 -17303.928,E2 -17303.928} C_VEL
LIN {X 0,Y 277.23,Z 280.766,A -85,B 0,C 180,E1 -17307.469,E2 -17307.469} C_VEL
LIN {X 0,Y 277.223,Z 280.765,A -85,B 0,C 180,E1 -17310.466,E2 -17310.466} C_VEL
LIN {X 0,Y 277.241,Z 280.765,A -85,B 0,C 180,E1 -17313.896,E2 -17313.896} C_VEL
LIN {X 0,Y 277.23,Z 280.768,A -85,B 0,C 180,E1 -17317.475,E2 -17317.475} C_VEL
LIN {X 0,Y 277.179,Z 280.774,A -85,B 0,C 180,E1 -17321.242,E2 -17321.242} C_VEL
LIN {X 0,Y 277.169,Z 280.775,A -85,B 0,C 180,E1 -17325.233,E2 -17325.233} C_VEL
LIN {X 0,Y 277.18,Z 280.772,A -85,B 0,C 180,E1 -17328.759,E2 -17328.759} C_VEL
LIN {X 0,Y 277.251,Z 280.762,A -85,B 0,C 180,E1 -17332.529,E2 -17332.529} C_VEL
LIN {X 0,Y 277.242,Z 280.762,A -85,B 0,C 180,E1 -17336.105,E2 -17336.105} C_VEL
LIN {X 0,Y 277.294,Z 280.935,A -85,B 0,C 180,E1 -17338.354,E2 -17338.354} C_VEL
LIN {X 0,Y 279.23,Z 290.327,A -85,B 0,C 180,E1 -17341.754,E2 -17341.754} C_VEL
LIN {X 0,Y 280.545,Z 297.975,A -85,B 0,C 180,E1 -17344.401,E2 -17344.401} C_VEL
LIN {X 0,Y 279.418,Z 306.831,A -85,B 0,C 180,E1 -17347.204,E2 -17347.204} C_VEL
LIN {X 0,Y 283.476,Z 333.727,A -85,B 0,C 180,E1 -17348.262,E2 -17348.262} C_VEL
LIN {X 0,Y 285.366,Z 352.02,A -85,B 0,C 180,E1 -17348.893,E2 -17348.893} C_VEL
LIN {X 0,Y 284.648,Z 385.756,A -85,B 0,C 180,E1 -17349.779,E2 -17349.779} C_VEL
LIN {X 0,Y 283.935,Z 396.693,A -85,B 0,C 180,E1 -17350.28,E2 -17350.28} C_VEL
LIN {X 0,Y 282.802,Z 408.585,A -85,B 0,C 180,E1 -17351.152,E2 -17351.152} C_VEL
LIN {X 0,Y 281.765,Z 417.283,A -85,B 0,C 180,E1 -17352.022,E2 -17352.022} C_VEL
LIN {X 0,Y 280.67,Z 425.599,A -85,B 0,C 180,E1 -17353.078,E2 -17353.078} C_VEL
LIN {X 0,Y 279.518,Z 433.477,A -85,B 0,C 180,E1 -17354.319,E2 -17354.319} C_VEL
LIN {X 0,Y 278.393,Z 440.851,A -85,B 0,C 180,E1 -17355.752,E2 -17355.752} C_VEL
LIN {X 0,Y 277.276,Z 448.342,A -85,B 0,C 180,E1 -17357.559,E2 -17357.559} C_VEL
LIN {X 0,Y 276.262,Z 455.189,A -85,B 0,C 180,E1 -17359.743,E2 -17359.743} C_VEL
LIN {X 0,Y 275.715,Z 460.406,A -85,B 0,C 180,E1 -17361.942,E2 -17361.942} C_VEL
LIN {X 0,Y 275.413,Z 464.242,A -85,B 0,C 180,E1 -17364.142,E2 -17364.142} C_VEL
LIN {X 0,Y 275.357,Z 466.009,A -85,B 0,C 180,E1 -17365.609,E2 -17365.609} C_VEL
LIN {X 0,Y 275.412,Z 467.279,A -85,B 0,C 180,E1 -17367.075,E2 -17367.075} C_VEL
LIN {X 0,Y 275.425,Z 468.066,A -85,B 0,C 180,E1 -17368.539,E2 -17368.539} C_VEL
LIN {X 0,Y 275.529,Z 468.368,A -85,B 0,C 180,E1 -17370.001,E2 -17370.001} C_VEL
LIN {X 0,Y 275.425,Z 468.059,A -85,B 0,C 180,E1 -17371.463,E2 -17371.463} C_VEL
LIN {X 0,Y 275.412,Z 467.259,A -85,B 0,C 180,E1 -17372.926,E2 -17372.926} C_VEL
LIN {X 0,Y 275.411,Z 464.568,A -85,B 0,C 180,E1 -17375.612,E2 -17375.612} C_VEL
LIN {X 0,Y 275.581,Z 461.839,A -85,B 0,C 180,E1 -17377.327,E2 -17377.327} C_VEL
LIN {X 0,Y 276.05,Z 457.041,A -85,B 0,C 180,E1 -17379.526,E2 -17379.526} C_VEL
LIN {X 0,Y 276.706,Z 451.856,A -85,B 0,C 180,E1 -17381.353,E2 -17381.353} C_VEL
LIN {X 0,Y 277.444,Z 446.796,A -85,B 0,C 180,E1 -17382.807,E2 -17382.807} C_VEL
LIN {X 0,Y 278.371,Z 440.709,A -85,B 0,C 180,E1 -17384.251,E2 -17384.251} C_VEL
LIN {X 0,Y 279.517,Z 433.311,A -85,B 0,C 180,E1 -17385.682,E2 -17385.682} C_VEL
LIN {X 0,Y 280.673,Z 425.393,A -85,B 0,C 180,E1 -17386.924,E2 -17386.924} C_VEL
LIN {X 0,Y 281.754,Z 417.027,A -85,B 0,C 180,E1 -17387.98,E2 -17387.98} C_VEL
LIN {X 0,Y 283.012,Z 406.245,A -85,B 0,C 180,E1 -17389.031,E2 -17389.031} C_VEL
LIN {X 0,Y 283.956,Z 395.105,A -85,B 0,C 180,E1 -17389.778,E2 -17389.778} C_VEL
LIN {X 0,Y 284.615,Z 385.605,A -85,B 0,C 180,E1 -17390.198,E2 -17390.198} C_VEL
LIN {X 0,Y 285.274,Z 350.016,A -85,B 0,C 180,E1 -17391.136,E2 -17391.136} C_VEL
LIN {X 0,Y 282.357,Z 325.98,A -85,B 0,C 180,E1 -17392.003,E2 -17392.003} C_VEL
LIN {X 0,Y 279.419,Z 306.744,A -85,B 0,C 180,E1 -17392.792,E2 -17392.792} C_VEL
LIN {X 0,Y 280.542,Z 297.88,A -85,B 0,C 180,E1 -17395.597,E2 -17395.597} C_VEL
LIN {X 0,Y 279.015,Z 289.25,A -85,B 0,C 180,E1 -17398.594,E2 -17398.594} C_VEL
LIN {X 0,Y 277.266,Z 280.756,A -85,B 0,C 180,E1 -17401.752,E2 -17401.752} C_VEL
LIN {X 0,Y 277.274,Z 280.758,A -85,B 0,C 180,E1 -17405.797,E2 -17405.797} C_VEL
LIN {X 0,Y 277.217,Z 280.767,A -85,B 0,C 180,E1 -17409.332,E2 -17409.332} C_VEL
LIN {X 0,Y 277.191,Z 280.771,A -85,B 0,C 180,E1 -17413.202,E2 -17413.202} C_VEL
LIN {X 0,Y 277.193,Z 280.769,A -85,B 0,C 180,E1 -17417.331,E2 -17417.331} C_VEL
LIN {X 0,Y 277.224,Z 280.765,A -85,B 0,C 180,E1 -17421.804,E2 -17421.804} C_VEL
LIN {X 0,Y 277.278,Z 280.761,A -85,B 0,C 180,E1 -17424.341,E2 -17424.341} C_VEL
LIN {X 0,Y 277.239,Z 280.763,A -85,B 0,C 180,E1 -17427.836,E2 -17427.836} C_VEL
LIN {X 0,Y 277.217,Z 280.764,A -85,B 0,C 180,E1 -17431.205,E2 -17431.205} C_VEL
LIN {X 0,Y 277.232,Z 280.764,A -85,B 0,C 180,E1 -17434.472,E2 -17434.472} C_VEL
LIN {X 0,Y 277.248,Z 280.762,A -85,B 0,C 180,E1 -17437.652,E2 -17437.652} C_VEL
LIN {X 0,Y 277.27,Z 280.758,A -85,B 0,C 180,E1 -17440.761,E2 -17440.761} C_VEL
LIN {X 0,Y 277.366,Z 280.745,A -85,B 0,C 180,E1 -17445.322,E2 -17445.322} C_VEL
LIN {X 0,Y 277.451,Z 280.73,A -85,B 0,C 180,E1 -17449.787,E2 -17449.787} C_VEL
LIN {X 0,Y 277.594,Z 280.705,A -85,B 0,C 180,E1 -17452.728,E2 -17452.728} C_VEL
LIN {X 0,Y 277.804,Z 280.691,A -85,B 0,C 180,E1 -17458.551,E2 -17458.551} C_VEL
LIN {X 0,Y 277.806,Z 280.686,A -85,B 0,C 180,E1 -17461.45,E2 -17461.45} C_VEL
LIN {X 0,Y 277.602,Z 280.717,A -85,B 0,C 180,E1 -17467.272,E2 -17467.272} C_VEL
LIN {X 0,Y 277.456,Z 280.734,A -85,B 0,C 180,E1 -17470.213,E2 -17470.213} C_VEL
LIN {X 0,Y 277.373,Z 280.736,A -85,B 0,C 180,E1 -17474.678,E2 -17474.678} C_VEL
LIN {X 0,Y 277.277,Z 280.758,A -85,B 0,C 180,E1 -17479.239,E2 -17479.239} C_VEL
LIN {X 0,Y 277.257,Z 280.757,A -85,B 0,C 180,E1 -17483.927,E2 -17483.927} C_VEL
LIN {X 0,Y 277.241,Z 280.759,A -85,B 0,C 180,E1 -17487.47,E2 -17487.47} C_VEL
LIN {X 0,Y 277.23,Z 280.766,A -85,B 0,C 180,E1 -17490.465,E2 -17490.465} C_VEL
LIN {X 0,Y 277.248,Z 280.756,A -85,B 0,C 180,E1 -17493.896,E2 -17493.896} C_VEL
LIN {X 0,Y 277.234,Z 280.761,A -85,B 0,C 180,E1 -17497.475,E2 -17497.475} C_VEL
LIN {X 0,Y 277.178,Z 280.767,A -85,B 0,C 180,E1 -17501.242,E2 -17501.242} C_VEL
LIN {X 0,Y 277.176,Z 280.771,A -85,B 0,C 180,E1 -17505.232,E2 -17505.232} C_VEL
LIN {X 0,Y 277.185,Z 280.764,A -85,B 0,C 180,E1 -17508.758,E2 -17508.758} C_VEL
LIN {X 0,Y 277.252,Z 280.745,A -85,B 0,C 180,E1 -17512.528,E2 -17512.528} C_VEL
LIN {X 0,Y 277.248,Z 280.763,A -85,B 0,C 180,E1 -17516.104,E2 -17516.104} C_VEL
LIN {X 0,Y 277.23,Z 280.766,A -85,B 0,C 180,E1 -17519.534,E2 -17519.534} C_VEL
LIN {X 0,Y 277.255,Z 280.761,A -85,B 0,C 180,E1 -17522.852,E2 -17522.852} C_VEL
LIN {X 0,Y 277.292,Z 280.761,A -85,B 0,C 180,E1 -17527.148,E2 -17527.148} C_VEL
LIN {X 0,Y 278.28,Z 283.589,A -85,B 0,C 180,E1 -17527.327,E2 -17527.327} C_VEL
LIN {X 0,Y 284.098,Z 297.335,A -85,B 0,C 180,E1 -17528.194,E2 -17528.194} C_VEL
LIN {X 0,Y 286.254,Z 303.708,A -85,B 0,C 180,E1 -17528.539,E2 -17528.539} C_VEL
LIN {X 0,Y 285.151,Z 355.389,A -85,B 0,C 180,E1 -17529.861,E2 -17529.861} C_VEL
LIN {X 0,Y 284.833,Z 365.145,A -85,B 0,C 180,E1 -17530.308,E2 -17530.308} C_VEL
LIN {X 0,Y 284.262,Z 376.198,A -85,B 0,C 180,E1 -17531.064,E2 -17531.064} C_VEL
LIN {X 0,Y 283.185,Z 386.99,A -85,B 0,C 180,E1 -17532.114,E2 -17532.114} C_VEL
LIN {X 0,Y 282.327,Z 394.136,A -85,B 0,C 180,E1 -17532.992,E2 -17532.992} C_VEL
LIN {X 0,Y 281.336,Z 402.237,A -85,B 0,C 180,E1 -17534.236,E2 -17534.236} C_VEL
LIN {X 0,Y 280.4,Z 408.918,A -85,B 0,C 180,E1 -17535.484,E2 -17535.484} C_VEL
LIN {X 0,Y 279.39,Z 415.245,A -85,B 0,C 180,E1 -17536.914,E2 -17536.914} C_VEL
LIN {X 0,Y 278.297,Z 421.666,A -85,B 0,C 180,E1 -17538.713,E2 -17538.713} C_VEL
LIN {X 0,Y 277.486,Z 426.782,A -85,B 0,C 180,E1 -17540.524,E2 -17540.524} C_VEL
LIN {X 0,Y 276.777,Z 431.509,A -85,B 0,C 180,E1 -17542.705,E2 -17542.705} C_VEL
LIN {X 0,Y 276.318,Z 433.819,A -85,B 0,C 180,E1 -17544.16,E2 -17544.16} C_VEL
LIN {X 0,Y 275.975,Z 435.575,A -85,B 0,C 180,E1 -17545.618,E2 -17545.618} C_VEL
LIN {X 0,Y 275.742,Z 436.839,A -85,B 0,C 180,E1 -17547.077,E2 -17547.077} C_VEL
LIN {X 0,Y 275.601,Z 437.636,A -85,B 0,C 180,E1 -17548.538,E2 -17548.538} C_VEL
LIN {X 0,Y 275.559,Z 437.94,A -85,B 0,C 180,E1 -17549.999,E2 -17549.999} C_VEL
LIN {X 0,Y 275.598,Z 437.663,A -85,B 0,C 180,E1 -17551.46,E2 -17551.46} C_VEL
LIN {X 0,Y 275.728,Z 436.919,A -85,B 0,C 180,E1 -17552.921,E2 -17552.921} C_VEL
LIN {X 0,Y 275.968,Z 435.708,A -85,B 0,C 180,E1 -17554.381,E2 -17554.381} C_VEL
LIN {X 0,Y 276.533,Z 432.867,A -85,B 0,C 180,E1 -17556.566,E2 -17556.566} C_VEL
LIN {X 0,Y 277.108,Z 429.378,A -85,B 0,C 180,E1 -17558.46,E2 -17558.46} C_VEL
LIN {X 0,Y 277.78,Z 425.201,A -85,B 0,C 180,E1 -17560.2,E2 -17560.2} C_VEL
LIN {X 0,Y 278.654,Z 419.729,A -85,B 0,C 180,E1 -17562.009,E2 -17562.009} C_VEL
LIN {X 0,Y 279.883,Z 412.837,A -85,B 0,C 180,E1 -17563.8,E2 -17563.8} C_VEL
LIN {X 0,Y 281.058,Z 404.926,A -85,B 0,C 180,E1 -17565.407,E2 -17565.407} C_VEL
LIN {X 0,Y 282.038,Z 397.38,A -85,B 0,C 180,E1 -17566.652,E2 -17566.652} C_VEL
LIN {X 0,Y 282.811,Z 390.958,A -85,B 0,C 180,E1 -17567.536,E2 -17567.536} C_VEL
LIN {X 0,Y 283.698,Z 383.143,A -85,B 0,C 180,E1 -17568.411,E2 -17568.411} C_VEL
LIN {X 0,Y 284.452,Z 374.18,A -85,B 0,C 180,E1 -17569.202,E2 -17569.202} C_VEL
LIN {X 0,Y 284.917,Z 364.823,A -85,B 0,C 180,E1 -17569.825,E2 -17569.825} C_VEL
LIN {X 0,Y 285.216,Z 355.426,A -85,B 0,C 180,E1 -17570.254,E2 -17570.254} C_VEL
LIN {X 0,Y 286.373,Z 303.979,A -85,B 0,C 180,E1 -17571.566,E2 -17571.566} C_VEL
LIN {X 0,Y 281.419,Z 290.642,A -85,B 0,C 180,E1 -17572.333,E2 -17572.333} C_VEL
LIN {X 0,Y 277.363,Z 281.199,A -85,B 0,C 180,E1 -17572.945,E2 -17572.945} C_VEL
LIN {X 0,Y 277.275,Z 280.763,A -85,B 0,C 180,E1 -17573.007,E2 -17573.007} C_VEL
LIN {X 0,Y 277.234,Z 280.764,A -85,B 0,C 180,E1 -17577.468,E2 -17577.468} C_VEL
LIN {X 0,Y 277.226,Z 280.767,A -85,B 0,C 180,E1 -17580.465,E2 -17580.465} C_VEL
LIN {X 0,Y 277.244,Z 280.763,A -85,B 0,C 180,E1 -17583.895,E2 -17583.895} C_VEL
LIN {X 0,Y 277.229,Z 280.762,A -85,B 0,C 180,E1 -17587.474,E2 -17587.474} C_VEL
LIN {X 0,Y 277.173,Z 280.764,A -85,B 0,C 180,E1 -17591.242,E2 -17591.242} C_VEL
LIN {X 0,Y 277.171,Z 280.77,A -85,B 0,C 180,E1 -17595.231,E2 -17595.231} C_VEL
LIN {X 0,Y 277.173,Z 280.764,A -85,B 0,C 180,E1 -17598.757,E2 -17598.757} C_VEL
LIN {X 0,Y 277.228,Z 280.761,A -85,B 0,C 180,E1 -17602.524,E2 -17602.524} C_VEL
LIN {X 0,Y 277.242,Z 280.761,A -85,B 0,C 180,E1 -17606.103,E2 -17606.103} C_VEL
LIN {X 0,Y 277.224,Z 280.766,A -85,B 0,C 180,E1 -17609.534,E2 -17609.534} C_VEL
LIN {X 0,Y 277.285,Z 280.753,A -85,B 0,C 180,E1 -17612.856,E2 -17612.856} C_VEL
LIN {X 0,Y 277.278,Z 280.756,A -85,B 0,C 180,E1 -17616.075,E2 -17616.075} C_VEL
LIN {X 0,Y 277.275,Z 280.758,A -85,B 0,C 180,E1 -17620.761,E2 -17620.761} C_VEL
LIN {X 0,Y 277.366,Z 280.736,A -85,B 0,C 180,E1 -17625.322,E2 -17625.322} C_VEL
LIN {X 0,Y 277.456,Z 280.734,A -85,B 0,C 180,E1 -17629.926,E2 -17629.926} C_VEL
LIN {X 0,Y 277.17,Z 280.773,A -85,B 0,C 180,E1 -17630.738,E2 -17630.738} C_VEL
LIN {X 0,Y 275.208,Z 281.015,A -85,B 0,C 180,E1 -17632.329,E2 -17632.329} C_VEL
LIN {X 0,Y 271.457,Z 281.474,A -85,B 0,C 180,E1 -17634.72,E2 -17634.72} C_VEL
LIN {X 0,Y 270.496,Z 281.589,A -85,B 0,C 180,E1 -17635.966,E2 -17635.966} C_VEL
LIN {X 0,Y 270.466,Z 281.591,A -85,B 0,C 180,E1 -17636.388,E2 -17636.388} C_VEL
LIN {X 0,Y 270.764,Z 281.562,A -85,B 0,C 180,E1 -17638.512,E2 -17638.512} C_VEL
LIN {X 0,Y 270.764,Z 281.568,A -85,B 0,C 180,E1 -17641.487,E2 -17641.487} C_VEL
LIN {X 0,Y 270.556,Z 281.594,A -85,B 0,C 180,E1 -17647.463,E2 -17647.463} C_VEL
LIN {X 0,Y 270.38,Z 281.616,A -85,B 0,C 180,E1 -17650.483,E2 -17650.483} C_VEL
LIN {X 0,Y 270.333,Z 281.62,A -85,B 0,C 180,E1 -17655.068,E2 -17655.068} C_VEL
LIN {X 0,Y 270.214,Z 281.639,A -85,B 0,C 180,E1 -17659.762,E2 -17659.762} C_VEL
LIN {X 0,Y 270.177,Z 281.64,A -85,B 0,C 180,E1 -17664.436,E2 -17664.436} C_VEL
LIN {X 0,Y 270.179,Z 281.645,A -85,B 0,C 180,E1 -17667.919,E2 -17667.919} C_VEL
LIN {X 0,Y 270.164,Z 281.647,A -85,B 0,C 180,E1 -17671.351,E2 -17671.351} C_VEL
LIN {X 0,Y 270.193,Z 281.642,A -85,B 0,C 180,E1 -17674.907,E2 -17674.907} C_VEL
LIN {X 0,Y 270.163,Z 281.645,A -85,B 0,C 180,E1 -17678.703,E2 -17678.703} C_VEL
LIN {X 0,Y 270.143,Z 281.651,A -85,B 0,C 180,E1 -17683.245,E2 -17683.245} C_VEL
LIN {X 0,Y 270.147,Z 281.648,A -85,B 0,C 180,E1 -17687.438,E2 -17687.438} C_VEL
LIN {X 0,Y 270.204,Z 281.641,A -85,B 0,C 180,E1 -17691.375,E2 -17691.375} C_VEL
LIN {X 0,Y 270.194,Z 281.642,A -85,B 0,C 180,E1 -17695.095,E2 -17695.095} C_VEL
LIN {X 0,Y 270.263,Z 281.788,A -85,B 0,C 180,E1 -17697.897,E2 -17697.897} C_VEL
LIN {X 0,Y 272.195,Z 291.143,A -85,B 0,C 180,E1 -17701.386,E2 -17701.386} C_VEL
LIN {X 0,Y 273.538,Z 298.757,A -85,B 0,C 180,E1 -17704.102,E2 -17704.102} C_VEL
LIN {X 0,Y 272.978,Z 303.57,A -85,B 0,C 180,E1 -17705.675,E2 -17705.675} C_VEL
LIN {X 0,Y 272.616,Z 306.372,A -85,B 0,C 180,E1 -17706.583,E2 -17706.583} C_VEL
LIN {X 0,Y 276.487,Z 331.692,A -85,B 0,C 180,E1 -17707.638,E2 -17707.638} C_VEL
LIN {X 0,Y 278.76,Z 351.983,A -85,B 0,C 180,E1 -17708.377,E2 -17708.377} C_VEL
LIN {X 0,Y 278.005,Z 385.38,A -85,B 0,C 180,E1 -17709.274,E2 -17709.274} C_VEL
LIN {X 0,Y 277.271,Z 396.077,A -85,B 0,C 180,E1 -17709.772,E2 -17709.772} C_VEL
LIN {X 0,Y 276.096,Z 408.199,A -85,B 0,C 180,E1 -17710.677,E2 -17710.677} C_VEL
LIN {X 0,Y 275.025,Z 416.895,A -85,B 0,C 180,E1 -17711.566,E2 -17711.566} C_VEL
LIN {X 0,Y 273.861,Z 425.209,A -85,B 0,C 180,E1 -17712.644,E2 -17712.644} C_VEL
LIN {X 0,Y 272.685,Z 433.088,A -85,B 0,C 180,E1 -17713.916,E2 -17713.916} C_VEL
LIN {X 0,Y 271.508,Z 440.461,A -85,B 0,C 180,E1 -17715.383,E2 -17715.383} C_VEL
LIN {X 0,Y 270.319,Z 447.951,A -85,B 0,C 180,E1 -17717.234,E2 -17717.234} C_VEL
LIN {X 0,Y 269.262,Z 454.797,A -85,B 0,C 180,E1 -17719.473,E2 -17719.473} C_VEL
LIN {X 0,Y 268.649,Z 460.013,A -85,B 0,C 180,E1 -17721.728,E2 -17721.728} C_VEL
LIN {X 0,Y 268.344,Z 463.85,A -85,B 0,C 180,E1 -17723.987,E2 -17723.987} C_VEL
LIN {X 0,Y 268.265,Z 465.617,A -85,B 0,C 180,E1 -17725.493,E2 -17725.493} C_VEL
LIN {X 0,Y 268.337,Z 466.889,A -85,B 0,C 180,E1 -17726.998,E2 -17726.998} C_VEL
LIN {X 0,Y 268.344,Z 467.675,A -85,B 0,C 180,E1 -17728.5,E2 -17728.5} C_VEL
LIN {X 0,Y 268.441,Z 467.977,A -85,B 0,C 180,E1 -17730.001,E2 -17730.001} C_VEL
LIN {X 0,Y 268.344,Z 467.668,A -85,B 0,C 180,E1 -17731.502,E2 -17731.502} C_VEL
LIN {X 0,Y 268.337,Z 466.868,A -85,B 0,C 180,E1 -17733.003,E2 -17733.003} C_VEL
LIN {X 0,Y 268.333,Z 464.409,A -85,B 0,C 180,E1 -17735.577,E2 -17735.577} C_VEL
LIN {X 0,Y 268.523,Z 461.445,A -85,B 0,C 180,E1 -17737.52,E2 -17737.52} C_VEL
LIN {X 0,Y 269.022,Z 456.646,A -85,B 0,C 180,E1 -17739.777,E2 -17739.777} C_VEL
LIN {X 0,Y 269.733,Z 451.461,A -85,B 0,C 180,E1 -17741.651,E2 -17741.651} C_VEL
LIN {X 0,Y 270.497,Z 446.4,A -85,B 0,C 180,E1 -17743.141,E2 -17743.141} C_VEL
LIN {X 0,Y 271.486,Z 440.314,A -85,B 0,C 180,E1 -17744.62,E2 -17744.62} C_VEL
LIN {X 0,Y 272.686,Z 432.916,A -85,B 0,C 180,E1 -17746.086,E2 -17746.086} C_VEL
LIN {X 0,Y 273.879,Z 424.997,A -85,B 0,C 180,E1 -17747.357,E2 -17747.357} C_VEL
LIN {X 0,Y 275.022,Z 416.631,A -85,B 0,C 180,E1 -17748.436,E2 -17748.436} C_VEL
LIN {X 0,Y 276.258,Z 406.231,A -85,B 0,C 180,E1 -17749.479,E2 -17749.479} C_VEL
LIN {X 0,Y 277.274,Z 394.882,A -85,B 0,C 180,E1 -17750.265,E2 -17750.265} C_VEL
LIN {X 0,Y 277.969,Z 385.45,A -85,B 0,C 180,E1 -17750.694,E2 -17750.694} C_VEL
LIN {X 0,Y 278.657,Z 350.824,A -85,B 0,C 180,E1 -17751.63,E2 -17751.63} C_VEL
LIN {X 0,Y 275.538,Z 325.129,A -85,B 0,C 180,E1 -17752.588,E2 -17752.588} C_VEL
LIN {X 0,Y 272.608,Z 306.347,A -85,B 0,C 180,E1 -17753.392,E2 -17753.392} C_VEL
LIN {X 0,Y 273.541,Z 298.648,A -85,B 0,C 180,E1 -17755.899,E2 -17755.899} C_VEL
LIN {X 0,Y 271.727,Z 288.798,A -85,B 0,C 180,E1 -17759.435,E2 -17759.435} C_VEL
LIN {X 0,Y 270.216,Z 281.633,A -85,B 0,C 180,E1 -17762.166,E2 -17762.166} C_VEL
LIN {X 0,Y 270.21,Z 281.64,A -85,B 0,C 180,E1 -17766.743,E2 -17766.743} C_VEL
LIN {X 0,Y 270.149,Z 281.647,A -85,B 0,C 180,E1 -17770.571,E2 -17770.571} C_VEL
LIN {X 0,Y 270.129,Z 281.652,A -85,B 0,C 180,E1 -17774.626,E2 -17774.626} C_VEL
LIN {X 0,Y 270.151,Z 281.646,A -85,B 0,C 180,E1 -17777.438,E2 -17777.438} C_VEL
LIN {X 0,Y 270.153,Z 281.646,A -85,B 0,C 180,E1 -17781.365,E2 -17781.365} C_VEL
LIN {X 0,Y 270.199,Z 281.64,A -85,B 0,C 180,E1 -17785.094,E2 -17785.094} C_VEL
LIN {X 0,Y 270.172,Z 281.643,A -85,B 0,C 180,E1 -17789.142,E2 -17789.142} C_VEL
LIN {X 0,Y 270.189,Z 281.642,A -85,B 0,C 180,E1 -17792.177,E2 -17792.177} C_VEL
LIN {X 0,Y 270.183,Z 281.64,A -85,B 0,C 180,E1 -17795.564,E2 -17795.564} C_VEL
LIN {X 0,Y 270.217,Z 281.639,A -85,B 0,C 180,E1 -17800.238,E2 -17800.238} C_VEL
LIN {X 0,Y 270.338,Z 281.62,A -85,B 0,C 180,E1 -17804.932,E2 -17804.932} C_VEL
LIN {X 0,Y 270.384,Z 281.613,A -85,B 0,C 180,E1 -17809.517,E2 -17809.517} C_VEL
LIN {X 0,Y 270.555,Z 281.581,A -85,B 0,C 180,E1 -17812.537,E2 -17812.537} C_VEL
LIN {X 0,Y 270.77,Z 281.567,A -85,B 0,C 180,E1 -17818.513,E2 -17818.513} C_VEL
LIN {X 0,Y 270.771,Z 281.561,A -85,B 0,C 180,E1 -17821.487,E2 -17821.487} C_VEL
LIN {X 0,Y 270.564,Z 281.595,A -85,B 0,C 180,E1 -17827.463,E2 -17827.463} C_VEL
LIN {X 0,Y 270.389,Z 281.615,A -85,B 0,C 180,E1 -17830.483,E2 -17830.483} C_VEL
LIN {X 0,Y 270.34,Z 281.609,A -85,B 0,C 180,E1 -17835.068,E2 -17835.068} C_VEL
LIN {X 0,Y 270.221,Z 281.635,A -85,B 0,C 180,E1 -17839.762,E2 -17839.762} C_VEL
LIN {X 0,Y 270.184,Z 281.641,A -85,B 0,C 180,E1 -17844.436,E2 -17844.436} C_VEL
LIN {X 0,Y 270.188,Z 281.638,A -85,B 0,C 180,E1 -17847.918,E2 -17847.918} C_VEL
LIN {X 0,Y 270.171,Z 281.641,A -85,B 0,C 180,E1 -17851.35,E2 -17851.35} C_VEL
LIN {X 0,Y 270.199,Z 281.63,A -85,B 0,C 180,E1 -17854.906,E2 -17854.906} C_VEL
LIN {X 0,Y 270.17,Z 281.644,A -85,B 0,C 180,E1 -17858.702,E2 -17858.702} C_VEL
LIN {X 0,Y 270.15,Z 281.64,A -85,B 0,C 180,E1 -17863.245,E2 -17863.245} C_VEL
LIN {X 0,Y 270.153,Z 281.646,A -85,B 0,C 180,E1 -17867.437,E2 -17867.437} C_VEL
LIN {X 0,Y 270.194,Z 281.62,A -85,B 0,C 180,E1 -17871.371,E2 -17871.371} C_VEL
LIN {X 0,Y 270.199,Z 281.637,A -85,B 0,C 180,E1 -17875.093,E2 -17875.093} C_VEL
LIN {X 0,Y 270.173,Z 281.643,A -85,B 0,C 180,E1 -17879.141,E2 -17879.141} C_VEL
LIN {X 0,Y 270.19,Z 281.642,A -85,B 0,C 180,E1 -17882.176,E2 -17882.176} C_VEL
LIN {X 0,Y 270.247,Z 281.639,A -85,B 0,C 180,E1 -17886.507,E2 -17886.507} C_VEL
LIN {X 0,Y 271.308,Z 284.604,A -85,B 0,C 180,E1 -17886.727,E2 -17886.727} C_VEL
LIN {X 0,Y 277.818,Z 299.808,A -85,B 0,C 180,E1 -17887.732,E2 -17887.732} C_VEL
LIN {X 0,Y 279.677,Z 305.171,A -85,B 0,C 180,E1 -17888.037,E2 -17888.037} C_VEL
LIN {X 0,Y 278.517,Z 355.797,A -85,B 0,C 180,E1 -17889.36,E2 -17889.36} C_VEL
LIN {X 0,Y 278.179,Z 365.547,A -85,B 0,C 180,E1 -17889.817,E2 -17889.817} C_VEL
LIN {X 0,Y 277.587,Z 376.596,A -85,B 0,C 180,E1 -17890.591,E2 -17890.591} C_VEL
LIN {X 0,Y 276.465,Z 387.386,A -85,B 0,C 180,E1 -17891.664,E2 -17891.664} C_VEL
LIN {X 0,Y 275.576,Z 394.53,A -85,B 0,C 180,E1 -17892.562,E2 -17892.562} C_VEL
LIN {X 0,Y 274.542,Z 402.63,A -85,B 0,C 180,E1 -17893.835,E2 -17893.835} C_VEL
LIN {X 0,Y 273.554,Z 409.312,A -85,B 0,C 180,E1 -17895.112,E2 -17895.112} C_VEL
LIN {X 0,Y 272.516,Z 415.637,A -85,B 0,C 180,E1 -17896.578,E2 -17896.578} C_VEL
LIN {X 0,Y 271.584,Z 420.894,A -85,B 0,C 180,E1 -17898.051,E2 -17898.051} C_VEL
LIN {X 0,Y 270.804,Z 425.279,A -85,B 0,C 180,E1 -17899.532,E2 -17899.532} C_VEL
LIN {X 0,Y 270.032,Z 429.888,A -85,B 0,C 180,E1 -17901.498,E2 -17901.498} C_VEL
LIN {X 0,Y 269.527,Z 433.068,A -85,B 0,C 180,E1 -17903.261,E2 -17903.261} C_VEL
LIN {X 0,Y 268.919,Z 435.966,A -85,B 0,C 180,E1 -17905.502,E2 -17905.502} C_VEL
LIN {X 0,Y 268.669,Z 437.23,A -85,B 0,C 180,E1 -17907,E2 -17907} C_VEL
LIN {X 0,Y 268.518,Z 438.028,A -85,B 0,C 180,E1 -17908.499,E2 -17908.499} C_VEL
LIN {X 0,Y 268.472,Z 438.331,A -85,B 0,C 180,E1 -17909.999,E2 -17909.999} C_VEL
LIN {X 0,Y 268.515,Z 438.054,A -85,B 0,C 180,E1 -17911.499,E2 -17911.499} C_VEL
LIN {X 0,Y 268.655,Z 437.31,A -85,B 0,C 180,E1 -17912.998,E2 -17912.998} C_VEL
LIN {X 0,Y 268.913,Z 436.098,A -85,B 0,C 180,E1 -17914.496,E2 -17914.496} C_VEL
LIN {X 0,Y 269.515,Z 433.256,A -85,B 0,C 180,E1 -17916.738,E2 -17916.738} C_VEL
LIN {X 0,Y 270.031,Z 430.132,A -85,B 0,C 180,E1 -17918.501,E2 -17918.501} C_VEL
LIN {X 0,Y 270.795,Z 425.592,A -85,B 0,C 180,E1 -17920.466,E2 -17920.466} C_VEL
LIN {X 0,Y 271.742,Z 420.117,A -85,B 0,C 180,E1 -17922.319,E2 -17922.319} C_VEL
LIN {X 0,Y 273.01,Z 413.226,A -85,B 0,C 180,E1 -17924.155,E2 -17924.155} C_VEL
LIN {X 0,Y 274.24,Z 405.313,A -85,B 0,C 180,E1 -17925.8,E2 -17925.8} C_VEL
LIN {X 0,Y 275.251,Z 397.767,A -85,B 0,C 180,E1 -17927.075,E2 -17927.075} C_VEL
LIN {X 0,Y 276.233,Z 389.85,A -85,B 0,C 180,E1 -17928.159,E2 -17928.159} C_VEL
LIN {X 0,Y 277.144,Z 381.662,A -85,B 0,C 180,E1 -17929.055,E2 -17929.055} C_VEL
LIN {X 0,Y 277.91,Z 373.354,A -85,B 0,C 180,E1 -17929.769,E2 -17929.769} C_VEL
LIN {X 0,Y 278.283,Z 364.375,A -85,B 0,C 180,E1 -17930.367,E2 -17930.367} C_VEL
LIN {X 0,Y 278.614,Z 355.144,A -85,B 0,C 180,E1 -17930.78,E2 -17930.78} C_VEL
LIN {X 0,Y 279.797,Z 305.474,A -85,B 0,C 180,E1 -17932.068,E2 -17932.068} C_VEL
LIN {X 0,Y 274.985,Z 292.813,A -85,B 0,C 180,E1 -17932.835,E2 -17932.835} C_VEL
LIN {X 0,Y 270.291,Z 282.085,A -85,B 0,C 180,E1 -17933.567,E2 -17933.567} C_VEL
LIN {X 0,Y 270.24,Z 281.636,A -85,B 0,C 180,E1 -17933.622,E2 -17933.622} C_VEL
LIN {X 0,Y 270.183,Z 281.643,A -85,B 0,C 180,E1 -17937.918,E2 -17937.918} C_VEL
LIN {X 0,Y 270.167,Z 281.643,A -85,B 0,C 180,E1 -17941.349,E2 -17941.349} C_VEL
LIN {X 0,Y 270.195,Z 281.638,A -85,B 0,C 180,E1 -17944.905,E2 -17944.905} C_VEL
LIN {X 0,Y 270.165,Z 281.644,A -85,B 0,C 180,E1 -17948.701,E2 -17948.701} C_VEL
LIN {X 0,Y 270.145,Z 281.643,A -85,B 0,C 180,E1 -17953.244,E2 -17953.244} C_VEL
LIN {X 0,Y 270.147,Z 281.64,A -85,B 0,C 180,E1 -17957.437,E2 -17957.437} C_VEL
LIN {X 0,Y 270.148,Z 281.645,A -85,B 0,C 180,E1 -17961.364,E2 -17961.364} C_VEL
LIN {X 0,Y 270.194,Z 281.638,A -85,B 0,C 180,E1 -17965.093,E2 -17965.093} C_VEL
LIN {X 0,Y 270.167,Z 281.642,A -85,B 0,C 180,E1 -17969.141,E2 -17969.141} C_VEL
LIN {X 0,Y 270.194,Z 281.636,A -85,B 0,C 180,E1 -17972.172,E2 -17972.172} C_VEL
LIN {X 0,Y 270.223,Z 281.637,A -85,B 0,C 180,E1 -17975.542,E2 -17975.542} C_VEL
LIN {X 0,Y 270.217,Z 281.636,A -85,B 0,C 180,E1 -17980.238,E2 -17980.238} C_VEL
LIN {X 0,Y 270.333,Z 281.611,A -85,B 0,C 180,E1 -17984.931,E2 -17984.931} C_VEL
LIN {X 0,Y 270.382,Z 281.616,A -85,B 0,C 180,E1 -17989.516,E2 -17989.516} C_VEL
LIN {X 0,Y 270.557,Z 281.595,A -85,B 0,C 180,E1 -17992.537,E2 -17992.537} C_VEL
LIN {X 0,Y 270.466,Z 281.591,A -85,B 0,C 180,E1 -17996.388,E2 -17996.388} C_VEL
LIN {X 0,Y 269.945,Z 281.662,A -85,B 0,C 180,E1 -17997.633,E2 -17997.633} C_VEL
LIN {X 0,Y 268.447,Z 281.854,A -85,B 0,C 180,E1 -17998.857,E2 -17998.857} C_VEL
LIN {X 0,Y 264.736,Z 282.319,A -85,B 0,C 180,E1 -18001.314,E2 -18001.314} C_VEL
LIN {X 0,Y 263.626,Z 282.46,A -85,B 0,C 180,E1 -18002.593,E2 -18002.593} C_VEL
LIN {X 0,Y 263.51,Z 282.471,A -85,B 0,C 180,E1 -18003.027,E2 -18003.027} C_VEL
LIN {X 0,Y 263.521,Z 282.471,A -85,B 0,C 180,E1 -18007.663,E2 -18007.663} C_VEL
LIN {X 0,Y 263.325,Z 282.493,A -85,B 0,C 180,E1 -18010.767,E2 -18010.767} C_VEL
LIN {X 0,Y 263.283,Z 282.499,A -85,B 0,C 180,E1 -18015.482,E2 -18015.482} C_VEL
LIN {X 0,Y 263.202,Z 282.511,A -85,B 0,C 180,E1 -18020.311,E2 -18020.311} C_VEL
LIN {X 0,Y 263.115,Z 282.52,A -85,B 0,C 180,E1 -18025.301,E2 -18025.301} C_VEL
LIN {X 0,Y 263.113,Z 282.522,A -85,B 0,C 180,E1 -18028.737,E2 -18028.737} C_VEL
LIN {X 0,Y 263.121,Z 282.522,A -85,B 0,C 180,E1 -18032.29,E2 -18032.29} C_VEL
LIN {X 0,Y 263.15,Z 282.52,A -85,B 0,C 180,E1 -18035.984,E2 -18035.984} C_VEL
LIN {X 0,Y 263.077,Z 282.529,A -85,B 0,C 180,E1 -18039.877,E2 -18039.877} C_VEL
LIN {X 0,Y 263.072,Z 282.528,A -85,B 0,C 180,E1 -18043.995,E2 -18043.995} C_VEL
LIN {X 0,Y 263.076,Z 282.527,A -85,B 0,C 180,E1 -18048.418,E2 -18048.418} C_VEL
LIN {X 0,Y 263.153,Z 282.517,A -85,B 0,C 180,E1 -18052.103,E2 -18052.103} C_VEL
LIN {X 0,Y 263.148,Z 282.518,A -85,B 0,C 180,E1 -18055.886,E2 -18055.886} C_VEL
LIN {X 0,Y 263.184,Z 282.568,A -85,B 0,C 180,E1 -18057.38,E2 -18057.38} C_VEL
LIN {X 0,Y 265.135,Z 292.006,A -85,B 0,C 180,E1 -18061.014,E2 -18061.014} C_VEL
LIN {X 0,Y 266.513,Z 299.326,A -85,B 0,C 180,E1 -18063.713,E2 -18063.713} C_VEL
LIN {X 0,Y 266.564,Z 301.257,A -85,B 0,C 180,E1 -18064.386,E2 -18064.386} C_VEL
LIN {X 0,Y 265.823,Z 305.983,A -85,B 0,C 180,E1 -18065.954,E2 -18065.954} C_VEL
LIN {X 0,Y 269.566,Z 330.074,A -85,B 0,C 180,E1 -18066.997,E2 -18066.997} C_VEL
LIN {X 0,Y 272.12,Z 351.754,A -85,B 0,C 180,E1 -18067.826,E2 -18067.826} C_VEL
LIN {X 0,Y 271.381,Z 385.004,A -85,B 0,C 180,E1 -18068.743,E2 -18068.743} C_VEL
LIN {X 0,Y 270.582,Z 396.31,A -85,B 0,C 180,E1 -18069.286,E2 -18069.286} C_VEL
LIN {X 0,Y 269.399,Z 407.812,A -85,B 0,C 180,E1 -18070.176,E2 -18070.176} C_VEL
LIN {X 0,Y 268.307,Z 416.508,A -85,B 0,C 180,E1 -18071.087,E2 -18071.087} C_VEL
LIN {X 0,Y 267.079,Z 424.82,A -85,B 0,C 180,E1 -18072.188,E2 -18072.188} C_VEL
LIN {X 0,Y 265.871,Z 432.699,A -85,B 0,C 180,E1 -18073.492,E2 -18073.492} C_VEL
LIN {X 0,Y 264.635,Z 440.071,A -85,B 0,C 180,E1 -18074.994,E2 -18074.994} C_VEL
LIN {X 0,Y 263.355,Z 447.558,A -85,B 0,C 180,E1 -18076.89,E2 -18076.89} C_VEL
LIN {X 0,Y 262.261,Z 454.405,A -85,B 0,C 180,E1 -18079.189,E2 -18079.189} C_VEL
LIN {X 0,Y 261.599,Z 459.62,A -85,B 0,C 180,E1 -18081.504,E2 -18081.504} C_VEL
LIN {X 0,Y 261.256,Z 463.458,A -85,B 0,C 180,E1 -18083.824,E2 -18083.824} C_VEL
LIN {X 0,Y 261.177,Z 465.225,A -85,B 0,C 180,E1 -18085.37,E2 -18085.37} C_VEL
LIN {X 0,Y 261.24,Z 466.497,A -85,B 0,C 180,E1 -18086.917,E2 -18086.917} C_VEL
LIN {X 0,Y 261.265,Z 467.284,A -85,B 0,C 180,E1 -18088.459,E2 -18088.459} C_VEL
LIN {X 0,Y 261.355,Z 467.585,A -85,B 0,C 180,E1 -18090.001,E2 -18090.001} C_VEL
LIN {X 0,Y 261.266,Z 467.277,A -85,B 0,C 180,E1 -18091.542,E2 -18091.542} C_VEL
LIN {X 0,Y 261.241,Z 466.475,A -85,B 0,C 180,E1 -18093.085,E2 -18093.085} C_VEL
LIN {X 0,Y 261.231,Z 464.281,A -85,B 0,C 180,E1 -18095.483,E2 -18095.483} C_VEL
LIN {X 0,Y 261.45,Z 461.05,A -85,B 0,C 180,E1 -18097.725,E2 -18097.725} C_VEL
LIN {X 0,Y 262.012,Z 456.251,A -85,B 0,C 180,E1 -18100.042,E2 -18100.042} C_VEL
LIN {X 0,Y 262.772,Z 451.067,A -85,B 0,C 180,E1 -18101.964,E2 -18101.964} C_VEL
LIN {X 0,Y 263.569,Z 446.005,A -85,B 0,C 180,E1 -18103.493,E2 -18103.493} C_VEL
LIN {X 0,Y 264.614,Z 439.919,A -85,B 0,C 180,E1 -18105.009,E2 -18105.009} C_VEL
LIN {X 0,Y 265.873,Z 432.521,A -85,B 0,C 180,E1 -18106.509,E2 -18106.509} C_VEL
LIN {X 0,Y 267.11,Z 424.601,A -85,B 0,C 180,E1 -18107.811,E2 -18107.811} C_VEL
LIN {X 0,Y 268.289,Z 416.234,A -85,B 0,C 180,E1 -18108.916,E2 -18108.916} C_VEL
LIN {X 0,Y 269.629,Z 405.542,A -85,B 0,C 180,E1 -18110.006,E2 -18110.006} C_VEL
LIN {X 0,Y 270.652,Z 394.402,A -85,B 0,C 180,E1 -18110.788,E2 -18110.788} C_VEL
LIN {X 0,Y 271.349,Z 385.121,A -85,B 0,C 180,E1 -18111.22,E2 -18111.22} C_VEL
LIN {X 0,Y 272.103,Z 353.113,A -85,B 0,C 180,E1 -18112.103,E2 -18112.103} C_VEL
LIN {X 0,Y 269.778,Z 331.969,A -85,B 0,C 180,E1 -18112.895,E2 -18112.895} C_VEL
LIN {X 0,Y 266.216,Z 308.5,A -85,B 0,C 180,E1 -18113.887,E2 -18113.887} C_VEL
LIN {X 0,Y 265.821,Z 305.936,A -85,B 0,C 180,E1 -18114.026,E2 -18114.026} C_VEL
LIN {X 0,Y 266.552,Z 301.177,A -85,B 0,C 180,E1 -18115.607,E2 -18115.607} C_VEL
LIN {X 0,Y 266.073,Z 296.976,A -85,B 0,C 180,E1 -18117.107,E2 -18117.107} C_VEL
LIN {X 0,Y 264.094,Z 286.819,A -85,B 0,C 180,E1 -18120.918,E2 -18120.918} C_VEL
LIN {X 0,Y 263.157,Z 282.513,A -85,B 0,C 180,E1 -18122.626,E2 -18122.626} C_VEL
LIN {X 0,Y 263.176,Z 282.516,A -85,B 0,C 180,E1 -18126.762,E2 -18126.762} C_VEL
LIN {X 0,Y 263.092,Z 282.525,A -85,B 0,C 180,E1 -18129.876,E2 -18129.876} C_VEL
LIN {X 0,Y 263.077,Z 282.527,A -85,B 0,C 180,E1 -18133.995,E2 -18133.995} C_VEL
LIN {X 0,Y 263.074,Z 282.53,A -85,B 0,C 180,E1 -18138.42,E2 -18138.42} C_VEL
LIN {X 0,Y 263.105,Z 282.525,A -85,B 0,C 180,E1 -18142.094,E2 -18142.094} C_VEL
LIN {X 0,Y 263.153,Z 282.518,A -85,B 0,C 180,E1 -18145.886,E2 -18145.886} C_VEL
LIN {X 0,Y 263.11,Z 282.523,A -85,B 0,C 180,E1 -18149.502,E2 -18149.502} C_VEL
LIN {X 0,Y 263.113,Z 282.522,A -85,B 0,C 180,E1 -18152.994,E2 -18152.994} C_VEL
LIN {X 0,Y 263.117,Z 282.524,A -85,B 0,C 180,E1 -18156.381,E2 -18156.381} C_VEL
LIN {X 0,Y 263.208,Z 282.511,A -85,B 0,C 180,E1 -18159.689,E2 -18159.689} C_VEL
LIN {X 0,Y 263.29,Z 282.499,A -85,B 0,C 180,E1 -18164.519,E2 -18164.519} C_VEL
LIN {X 0,Y 263.328,Z 282.492,A -85,B 0,C 180,E1 -18169.233,E2 -18169.233} C_VEL
LIN {X 0,Y 263.516,Z 282.457,A -85,B 0,C 180,E1 -18172.337,E2 -18172.337} C_VEL
LIN {X 0,Y 263.733,Z 282.443,A -85,B 0,C 180,E1 -18178.473,E2 -18178.473} C_VEL
LIN {X 0,Y 263.735,Z 282.436,A -85,B 0,C 180,E1 -18181.527,E2 -18181.527} C_VEL
LIN {X 0,Y 263.528,Z 282.47,A -85,B 0,C 180,E1 -18187.663,E2 -18187.663} C_VEL
LIN {X 0,Y 263.334,Z 282.495,A -85,B 0,C 180,E1 -18190.767,E2 -18190.767} C_VEL
LIN {X 0,Y 263.29,Z 282.487,A -85,B 0,C 180,E1 -18195.482,E2 -18195.482} C_VEL
LIN {X 0,Y 263.209,Z 282.51,A -85,B 0,C 180,E1 -18200.311,E2 -18200.311} C_VEL
LIN {X 0,Y 263.123,Z 282.52,A -85,B 0,C 180,E1 -18205.3,E2 -18205.3} C_VEL
LIN {X 0,Y 263.121,Z 282.521,A -85,B 0,C 180,E1 -18208.737,E2 -18208.737} C_VEL
LIN {X 0,Y 263.128,Z 282.52,A -85,B 0,C 180,E1 -18212.289,E2 -18212.289} C_VEL
LIN {X 0,Y 263.155,Z 282.508,A -85,B 0,C 180,E1 -18215.983,E2 -18215.983} C_VEL
LIN {X 0,Y 263.074,Z 282.529,A -85,B 0,C 180,E1 -18219.878,E2 -18219.878} C_VEL
LIN {X 0,Y 263.078,Z 282.524,A -85,B 0,C 180,E1 -18223.994,E2 -18223.994} C_VEL
LIN {X 0,Y 263.082,Z 282.522,A -85,B 0,C 180,E1 -18228.417,E2 -18228.417} C_VEL
LIN {X 0,Y 263.132,Z 282.497,A -85,B 0,C 180,E1 -18232.098,E2 -18232.098} C_VEL
LIN {X 0,Y 263.154,Z 282.52,A -85,B 0,C 180,E1 -18235.885,E2 -18235.885} C_VEL
LIN {X 0,Y 263.111,Z 282.524,A -85,B 0,C 180,E1 -18239.501,E2 -18239.501} C_VEL
LIN {X 0,Y 263.119,Z 282.523,A -85,B 0,C 180,E1 -18242.994,E2 -18242.994} C_VEL
LIN {X 0,Y 263.221,Z 282.657,A -85,B 0,C 180,E1 -18245.895,E2 -18245.895} C_VEL
LIN {X 0,Y 264.344,Z 285.581,A -85,B 0,C 180,E1 -18246.091,E2 -18246.091} C_VEL
LIN {X 0,Y 271.529,Z 302.115,A -85,B 0,C 180,E1 -18247.241,E2 -18247.241} C_VEL
LIN {X 0,Y 273.175,Z 307.244,A -85,B 0,C 180,E1 -18247.533,E2 -18247.533} C_VEL
LIN {X 0,Y 271.898,Z 356.206,A -85,B 0,C 180,E1 -18248.834,E2 -18248.834} C_VEL
LIN {X 0,Y 271.549,Z 365.949,A -85,B 0,C 180,E1 -18249.301,E2 -18249.301} C_VEL
LIN {X 0,Y 270.928,Z 376.994,A -85,B 0,C 180,E1 -18250.094,E2 -18250.094} C_VEL
LIN {X 0,Y 269.757,Z 387.781,A -85,B 0,C 180,E1 -18251.191,E2 -18251.191} C_VEL
LIN {X 0,Y 268.837,Z 394.925,A -85,B 0,C 180,E1 -18252.11,E2 -18252.11} C_VEL
LIN {X 0,Y 267.751,Z 403.025,A -85,B 0,C 180,E1 -18253.414,E2 -18253.414} C_VEL
LIN {X 0,Y 266.726,Z 409.705,A -85,B 0,C 180,E1 -18254.722,E2 -18254.722} C_VEL
LIN {X 0,Y 265.649,Z 416.03,A -85,B 0,C 180,E1 -18256.225,E2 -18256.225} C_VEL
LIN {X 0,Y 264.666,Z 421.287,A -85,B 0,C 180,E1 -18257.734,E2 -18257.734} C_VEL
LIN {X 0,Y 263.844,Z 425.672,A -85,B 0,C 180,E1 -18259.253,E2 -18259.253} C_VEL
LIN {X 0,Y 262.981,Z 430.57,A -85,B 0,C 180,E1 -18261.418,E2 -18261.418} C_VEL
LIN {X 0,Y 262.491,Z 433.461,A -85,B 0,C 180,E1 -18263.079,E2 -18263.079} C_VEL
LIN {X 0,Y 261.868,Z 436.357,A -85,B 0,C 180,E1 -18265.381,E2 -18265.381} C_VEL
LIN {X 0,Y 261.598,Z 437.622,A -85,B 0,C 180,E1 -18266.919,E2 -18266.919} C_VEL
LIN {X 0,Y 261.436,Z 438.419,A -85,B 0,C 180,E1 -18268.459,E2 -18268.459} C_VEL
LIN {X 0,Y 261.388,Z 438.722,A -85,B 0,C 180,E1 -18269.999,E2 -18269.999} C_VEL
LIN {X 0,Y 261.433,Z 438.445,A -85,B 0,C 180,E1 -18271.54,E2 -18271.54} C_VEL
LIN {X 0,Y 261.585,Z 437.7,A -85,B 0,C 180,E1 -18273.079,E2 -18273.079} C_VEL
LIN {X 0,Y 261.861,Z 436.488,A -85,B 0,C 180,E1 -18274.617,E2 -18274.617} C_VEL
LIN {X 0,Y 262.476,Z 433.646,A -85,B 0,C 180,E1 -18276.92,E2 -18276.92} C_VEL
